LIN {X 0,Y 382.745,Z 469.054,A -85,B 0,C 180,E1 -14676.834,E2 -14676.834} C_VEL
LIN {X 0,Y 379.922,Z 466.3,A -85,B 0,C 180,E1 -14678.454,E2 -14678.454} C_VEL
LIN {X 0,Y 378.17,Z 464.212,A -85,B 0,C 180,E1 -14679.366,E2 -14679.366} C_VEL
LIN {X 0,Y 375.017,Z 462.339,A -85,B 0,C 180,E1 -14680.642,E2 -14680.642} C_VEL
LIN {X 0,Y 371.721,Z 459.429,A -85,B 0,C 180,E1 -14681.895,E2 -14681.895} C_VEL
LIN {X 0,Y 368.971,Z 456.558,A -85,B 0,C 180,E1 -14682.858,E2 -14682.858} C_VEL
LIN {X 0,Y 365.379,Z 453.694,A -85,B 0,C 180,E1 -14683.945,E2 -14683.945} C_VEL
LIN {X 0,Y 361.344,Z 449.449,A -85,B 0,C 180,E1 -14685.108,E2 -14685.108} C_VEL
LIN {X 0,Y 357.38,Z 445.807,A -85,B 0,C 180,E1 -14686.135,E2 -14686.135} C_VEL
LIN {X 0,Y 354.585,Z 442.813,A -85,B 0,C 180,E1 -14686.804,E2 -14686.804} C_VEL
LIN {X 0,Y 351.005,Z 439.151,A -85,B 0,C 180,E1 -14687.633,E2 -14687.633} C_VEL
LIN {X 0,Y 348.399,Z 436.221,A -85,B 0,C 180,E1 -14688.218,E2 -14688.218} C_VEL
LIN {X 0,Y 345.155,Z 432.375,A -85,B 0,C 180,E1 -14688.921,E2 -14688.921} C_VEL
LIN {X 0,Y 341.006,Z 427.451,A -85,B 0,C 180,E1 -14689.766,E2 -14689.766} C_VEL
LIN {X 0,Y 339.453,Z 425.497,A -85,B 0,C 180,E1 -14690.077,E2 -14690.077} C_VEL
LIN {X 0,Y 337.07,Z 422.222,A -85,B 0,C 180,E1 -14690.545,E2 -14690.545} C_VEL
LIN {X 0,Y 336.014,Z 420.806,A -85,B 0,C 180,E1 -14690.746,E2 -14690.746} C_VEL
LIN {X 0,Y 334.263,Z 418.461,A -85,B 0,C 180,E1 -14691.08,E2 -14691.08} C_VEL
LIN {X 0,Y 333.682,Z 416.42,A -85,B 0,C 180,E1 -14691.257,E2 -14691.257} C_VEL
LIN {X 0,Y 333.715,Z 416.415,A -85,B 0,C 180,E1 -14695.101,E2 -14695.101} C_VEL
LIN {X 0,Y 333.717,Z 416.414,A -85,B 0,C 180,E1 -14697.811,E2 -14697.811} C_VEL
LIN {X 0,Y 333.693,Z 416.42,A -85,B 0,C 180,E1 -14700.362,E2 -14700.362} C_VEL
LIN {X 0,Y 333.681,Z 416.42,A -85,B 0,C 180,E1 -14704.774,E2 -14704.774} C_VEL
LIN {X 0,Y 333.678,Z 416.42,A -85,B 0,C 180,E1 -14708.805,E2 -14708.805} C_VEL
LIN {X 0,Y 333.686,Z 416.421,A -85,B 0,C 180,E1 -14712.511,E2 -14712.511} C_VEL
LIN {X 0,Y 333.63,Z 416.426,A -85,B 0,C 180,E1 -14715.962,E2 -14715.962} C_VEL
LIN {X 0,Y 333.643,Z 416.422,A -85,B 0,C 180,E1 -14719.316,E2 -14719.316} C_VEL
LIN {X 0,Y 333.663,Z 416.419,A -85,B 0,C 180,E1 -14723.168,E2 -14723.168} C_VEL
LIN {X 0,Y 333.638,Z 416.423,A -85,B 0,C 180,E1 -14726.793,E2 -14726.793} C_VEL
LIN {X 0,Y 333.7,Z 416.417,A -85,B 0,C 180,E1 -14729.71,E2 -14729.71} C_VEL
LIN {X 0,Y 333.74,Z 416.412,A -85,B 0,C 180,E1 -14732.402,E2 -14732.402} C_VEL
LIN {X 0,Y 333.723,Z 416.411,A -85,B 0,C 180,E1 -14735.091,E2 -14735.091} C_VEL
LIN {X 0,Y 333.678,Z 416.417,A -85,B 0,C 180,E1 -14739.02,E2 -14739.02} C_VEL
LIN {X 0,Y 333.701,Z 416.414,A -85,B 0,C 180,E1 -14739.93,E2 -14739.93} C_VEL
LIN {X 0,Y 333.092,Z 416.492,A -85,B 0,C 180,E1 -14740.937,E2 -14740.937} C_VEL
LIN {X 0,Y 330.267,Z 416.843,A -85,B 0,C 180,E1 -14742.576,E2 -14742.576} C_VEL
LIN {X 0,Y 327.851,Z 417.148,A -85,B 0,C 180,E1 -14743.904,E2 -14743.904} C_VEL
LIN {X 0,Y 326.828,Z 417.27,A -85,B 0,C 180,E1 -14744.932,E2 -14744.932} C_VEL
LIN {X 0,Y 326.754,Z 417.28,A -85,B 0,C 180,E1 -14745.28,E2 -14745.28} C_VEL
LIN {X 0,Y 326.766,Z 417.278,A -85,B 0,C 180,E1 -14748.84,E2 -14748.84} C_VEL
LIN {X 0,Y 326.976,Z 417.253,A -85,B 0,C 180,E1 -14752.591,E2 -14752.591} C_VEL
LIN {X 0,Y 326.775,Z 417.277,A -85,B 0,C 180,E1 -14755.066,E2 -14755.066} C_VEL
LIN {X 0,Y 327.045,Z 417.244,A -85,B 0,C 180,E1 -14757.537,E2 -14757.537} C_VEL
LIN {X 0,Y 327.196,Z 417.226,A -85,B 0,C 180,E1 -14760.001,E2 -14760.001} C_VEL
LIN {X 0,Y 327.045,Z 417.244,A -85,B 0,C 180,E1 -14762.464,E2 -14762.464} C_VEL
LIN {X 0,Y 326.994,Z 417.251,A -85,B 0,C 180,E1 -14766.17,E2 -14766.17} C_VEL
LIN {X 0,Y 326.913,Z 417.261,A -85,B 0,C 180,E1 -14768.656,E2 -14768.656} C_VEL
LIN {X 0,Y 326.732,Z 417.283,A -85,B 0,C 180,E1 -14772.422,E2 -14772.422} C_VEL
LIN {X 0,Y 326.753,Z 417.282,A -85,B 0,C 180,E1 -14774.958,E2 -14774.958} C_VEL
LIN {X 0,Y 326.731,Z 417.285,A -85,B 0,C 180,E1 -14778.839,E2 -14778.839} C_VEL
LIN {X 0,Y 326.62,Z 417.299,A -85,B 0,C 180,E1 -14782.788,E2 -14782.788} C_VEL
LIN {X 0,Y 326.689,Z 417.291,A -85,B 0,C 180,E1 -14785.484,E2 -14785.484} C_VEL
LIN {X 0,Y 326.647,Z 417.297,A -85,B 0,C 180,E1 -14789.661,E2 -14789.661} C_VEL
LIN {X 0,Y 326.607,Z 417.301,A -85,B 0,C 180,E1 -14794.02,E2 -14794.02} C_VEL
LIN {X 0,Y 326.687,Z 417.697,A -85,B 0,C 180,E1 -14795.511,E2 -14795.511} C_VEL
LIN {X 0,Y 327.062,Z 420.418,A -85,B 0,C 180,E1 -14799.324,E2 -14799.324} C_VEL
LIN {X 0,Y 327.357,Z 422.259,A -85,B 0,C 180,E1 -14801.724,E2 -14801.724} C_VEL
LIN {X 0,Y 327.716,Z 424.981,A -85,B 0,C 180,E1 -14805.049,E2 -14805.049} C_VEL
LIN {X 0,Y 327.837,Z 427.974,A -85,B 0,C 180,E1 -14808.352,E2 -14808.352} C_VEL
LIN {X 0,Y 327.499,Z 431.094,A -85,B 0,C 180,E1 -14811.514,E2 -14811.514} C_VEL
LIN {X 0,Y 327.027,Z 434.493,A -85,B 0,C 180,E1 -14814.751,E2 -14814.751} C_VEL
LIN {X 0,Y 326.606,Z 437.456,A -85,B 0,C 180,E1 -14817.456,E2 -14817.456} C_VEL
LIN {X 0,Y 326.204,Z 440.67,A -85,B 0,C 180,E1 -14820.295,E2 -14820.295} C_VEL
LIN {X 0,Y 325.882,Z 443.915,A -85,B 0,C 180,E1 -14823.071,E2 -14823.071} C_VEL
LIN {X 0,Y 325.607,Z 447.183,A -85,B 0,C 180,E1 -14825.789,E2 -14825.789} C_VEL
LIN {X 0,Y 325.418,Z 449.412,A -85,B 0,C 180,E1 -14827.655,E2 -14827.655} C_VEL
LIN {X 0,Y 327.712,Z 459.083,A -85,B 0,C 180,E1 -14828.196,E2 -14828.196} C_VEL
LIN {X 0,Y 329.534,Z 468.228,A -85,B 0,C 180,E1 -14828.81,E2 -14828.81} C_VEL
LIN {X 0,Y 331.05,Z 477.851,A -85,B 0,C 180,E1 -14829.573,E2 -14829.573} C_VEL
LIN {X 0,Y 332.004,Z 486.455,A -85,B 0,C 180,E1 -14830.364,E2 -14830.364} C_VEL
LIN {X 0,Y 332.422,Z 491.382,A -85,B 0,C 180,E1 -14830.871,E2 -14830.871} C_VEL
LIN {X 0,Y 330.921,Z 503.575,A -85,B 0,C 180,E1 -14832.224,E2 -14832.224} C_VEL
LIN {X 0,Y 329.776,Z 512.454,A -85,B 0,C 180,E1 -14833.467,E2 -14833.467} C_VEL
LIN {X 0,Y 328.719,Z 520.466,A -85,B 0,C 180,E1 -14834.817,E2 -14834.817} C_VEL
LIN {X 0,Y 327.875,Z 526.671,A -85,B 0,C 180,E1 -14836.046,E2 -14836.046} C_VEL
LIN {X 0,Y 326.889,Z 533.209,A -85,B 0,C 180,E1 -14837.585,E2 -14837.585} C_VEL
LIN {X 0,Y 326.349,Z 537.716,A -85,B 0,C 180,E1 -14838.824,E2 -14838.824} C_VEL
LIN {X 0,Y 325.644,Z 543.21,A -85,B 0,C 180,E1 -14840.685,E2 -14840.685} C_VEL
LIN {X 0,Y 325.21,Z 547.538,A -85,B 0,C 180,E1 -14842.55,E2 -14842.55} C_VEL
LIN {X 0,Y 324.998,Z 550.39,A -85,B 0,C 180,E1 -14844.125,E2 -14844.125} C_VEL
LIN {X 0,Y 324.911,Z 553.099,A -85,B 0,C 180,E1 -14846.279,E2 -14846.279} C_VEL
LIN {X 0,Y 324.837,Z 554.158,A -85,B 0,C 180,E1 -14847.52,E2 -14847.52} C_VEL
LIN {X 0,Y 324.815,Z 554.747,A -85,B 0,C 180,E1 -14848.76,E2 -14848.76} C_VEL
LIN {X 0,Y 324.815,Z 554.747,A -85,B 0,C 180,E1 -14851.24,E2 -14851.24} C_VEL
LIN {X 0,Y 324.837,Z 554.158,A -85,B 0,C 180,E1 -14852.48,E2 -14852.48} C_VEL
LIN {X 0,Y 324.93,Z 551.71,A -85,B 0,C 180,E1 -14854.963,E2 -14854.963} C_VEL
LIN {X 0,Y 325.121,Z 548.758,A -85,B 0,C 180,E1 -14856.828,E2 -14856.828} C_VEL
LIN {X 0,Y 325.474,Z 544.766,A -85,B 0,C 180,E1 -14858.693,E2 -14858.693} C_VEL
LIN {X 0,Y 326.08,Z 539.634,A -85,B 0,C 180,E1 -14860.556,E2 -14860.556} C_VEL
LIN {X 0,Y 326.735,Z 534.368,A -85,B 0,C 180,E1 -14862.106,E2 -14862.106} C_VEL
LIN {X 0,Y 327.648,Z 528.05,A -85,B 0,C 180,E1 -14863.647,E2 -14863.647} C_VEL
LIN {X 0,Y 328.457,Z 522.096,A -85,B 0,C 180,E1 -14864.878,E2 -14864.878} C_VEL
LIN {X 0,Y 329.441,Z 515.168,A -85,B 0,C 180,E1 -14866.1,E2 -14866.1} C_VEL
LIN {X 0,Y 330.455,Z 506.983,A -85,B 0,C 180,E1 -14867.322,E2 -14867.322} C_VEL
LIN {X 0,Y 331.552,Z 498.472,A -85,B 0,C 180,E1 -14868.379,E2 -14868.379} C_VEL
LIN {X 0,Y 332.416,Z 491.388,A -85,B 0,C 180,E1 -14869.129,E2 -14869.129} C_VEL
LIN {X 0,Y 331.654,Z 482.381,A -85,B 0,C 180,E1 -14870.027,E2 -14870.027} C_VEL
LIN {X 0,Y 330.019,Z 471.038,A -85,B 0,C 180,E1 -14870.981,E2 -14870.981} C_VEL
LIN {X 0,Y 328.019,Z 460.532,A -85,B 0,C 180,E1 -14871.714,E2 -14871.714} C_VEL
LIN {X 0,Y 325.445,Z 449.866,A -85,B 0,C 180,E1 -14872.326,E2 -14872.326} C_VEL
LIN {X 0,Y 325.417,Z 449.413,A -85,B 0,C 180,E1 -14872.344,E2 -14872.344} C_VEL
LIN {X 0,Y 325.738,Z 445.556,A -85,B 0,C 180,E1 -14875.563,E2 -14875.563} C_VEL
LIN {X 0,Y 326.06,Z 442.285,A -85,B 0,C 180,E1 -14878.306,E2 -14878.306} C_VEL
LIN {X 0,Y 326.604,Z 437.433,A -85,B 0,C 180,E1 -14882.544,E2 -14882.544} C_VEL
LIN {X 0,Y 327.052,Z 434.248,A -85,B 0,C 180,E1 -14885.464,E2 -14885.464} C_VEL
LIN {X 0,Y 327.496,Z 431.094,A -85,B 0,C 180,E1 -14888.486,E2 -14888.486} C_VEL
LIN {X 0,Y 327.828,Z 427.973,A -85,B 0,C 180,E1 -14891.649,E2 -14891.649} C_VEL
LIN {X 0,Y 327.834,Z 426.427,A -85,B 0,C 180,E1 -14893.314,E2 -14893.314} C_VEL
LIN {X 0,Y 327.49,Z 423.385,A -85,B 0,C 180,E1 -14896.855,E2 -14896.855} C_VEL
LIN {X 0,Y 327.142,Z 421.004,A -85,B 0,C 180,E1 -14899.872,E2 -14899.872} C_VEL
LIN {X 0,Y 326.816,Z 418.723,A -85,B 0,C 180,E1 -14902.977,E2 -14902.977} C_VEL
LIN {X 0,Y 326.67,Z 417.471,A -85,B 0,C 180,E1 -14904.837,E2 -14904.837} C_VEL
LIN {X 0,Y 326.613,Z 417.301,A -85,B 0,C 180,E1 -14907.455,E2 -14907.455} C_VEL
LIN {X 0,Y 326.659,Z 417.295,A -85,B 0,C 180,E1 -14910.34,E2 -14910.34} C_VEL
LIN {X 0,Y 326.687,Z 417.293,A -85,B 0,C 180,E1 -14914.515,E2 -14914.515} C_VEL
LIN {X 0,Y 326.644,Z 417.299,A -85,B 0,C 180,E1 -14918.544,E2 -14918.544} C_VEL
LIN {X 0,Y 326.741,Z 417.284,A -85,B 0,C 180,E1 -14921.177,E2 -14921.177} C_VEL
LIN {X 0,Y 326.759,Z 417.28,A -85,B 0,C 180,E1 -14925.432,E2 -14925.432} C_VEL
LIN {X 0,Y 326.765,Z 417.282,A -85,B 0,C 180,E1 -14928.838,E2 -14928.838} C_VEL
LIN {X 0,Y 326.972,Z 417.258,A -85,B 0,C 180,E1 -14932.59,E2 -14932.59} C_VEL
LIN {X 0,Y 326.774,Z 417.279,A -85,B 0,C 180,E1 -14935.064,E2 -14935.064} C_VEL
LIN {X 0,Y 327.043,Z 417.244,A -85,B 0,C 180,E1 -14937.536,E2 -14937.536} C_VEL
LIN {X 0,Y 327.193,Z 417.226,A -85,B 0,C 180,E1 -14939.999,E2 -14939.999} C_VEL
LIN {X 0,Y 327.042,Z 417.244,A -85,B 0,C 180,E1 -14942.463,E2 -14942.463} C_VEL
LIN {X 0,Y 326.965,Z 417.254,A -85,B 0,C 180,E1 -14946.663,E2 -14946.663} C_VEL
LIN {X 0,Y 326.807,Z 417.275,A -85,B 0,C 180,E1 -14949.906,E2 -14949.906} C_VEL
LIN {X 0,Y 326.753,Z 417.282,A -85,B 0,C 180,E1 -14953.685,E2 -14953.685} C_VEL
LIN {X 0,Y 326.693,Z 417.289,A -85,B 0,C 180,E1 -14957.527,E2 -14957.527} C_VEL
LIN {X 0,Y 326.658,Z 417.296,A -85,B 0,C 180,E1 -14960.134,E2 -14960.134} C_VEL
LIN {X 0,Y 326.645,Z 417.297,A -85,B 0,C 180,E1 -14964.129,E2 -14964.129} C_VEL
LIN {X 0,Y 326.679,Z 417.29,A -85,B 0,C 180,E1 -14966.857,E2 -14966.857} C_VEL
LIN {X 0,Y 326.635,Z 417.295,A -85,B 0,C 180,E1 -14970.612,E2 -14970.612} C_VEL
LIN {X 0,Y 326.602,Z 417.303,A -85,B 0,C 180,E1 -14974.019,E2 -14974.019} C_VEL
LIN {X 0,Y 326.624,Z 417.297,A -85,B 0,C 180,E1 -14977.239,E2 -14977.239} C_VEL
LIN {X 0,Y 326.629,Z 417.297,A -85,B 0,C 180,E1 -14980.202,E2 -14980.202} C_VEL
LIN {X 0,Y 326.651,Z 417.296,A -85,B 0,C 180,E1 -14983.51,E2 -14983.51} C_VEL
LIN {X 0,Y 326.645,Z 417.295,A -85,B 0,C 180,E1 -14987.014,E2 -14987.014} C_VEL
LIN {X 0,Y 326.639,Z 417.295,A -85,B 0,C 180,E1 -14990.766,E2 -14990.766} C_VEL
LIN {X 0,Y 326.607,Z 417.299,A -85,B 0,C 180,E1 -14994.481,E2 -14994.481} C_VEL
LIN {X 0,Y 326.602,Z 417.305,A -85,B 0,C 180,E1 -14997.456,E2 -14997.456} C_VEL
LIN {X 0,Y 326.655,Z 417.293,A -85,B 0,C 180,E1 -15000.341,E2 -15000.341} C_VEL
LIN {X 0,Y 326.685,Z 417.29,A -85,B 0,C 180,E1 -15004.517,E2 -15004.517} C_VEL
LIN {X 0,Y 326.696,Z 417.417,A -85,B 0,C 180,E1 -15007.846,E2 -15007.846} C_VEL
LIN {X 0,Y 327.662,Z 420.137,A -85,B 0,C 180,E1 -15008.038,E2 -15008.038} C_VEL
LIN {X 0,Y 329.517,Z 422.658,A -85,B 0,C 180,E1 -15008.363,E2 -15008.363} C_VEL
LIN {X 0,Y 331.952,Z 426.11,A -85,B 0,C 180,E1 -15008.797,E2 -15008.797} C_VEL
LIN {X 0,Y 335.942,Z 431.227,A -85,B 0,C 180,E1 -15009.532,E2 -15009.532} C_VEL
LIN {X 0,Y 340.414,Z 436.618,A -85,B 0,C 180,E1 -15010.402,E2 -15010.402} C_VEL
LIN {X 0,Y 345.474,Z 442.37,A -85,B 0,C 180,E1 -15011.446,E2 -15011.446} C_VEL
LIN {X 0,Y 350.954,Z 448.276,A -85,B 0,C 180,E1 -15012.679,E2 -15012.679} C_VEL
LIN {X 0,Y 353.634,Z 450.976,A -85,B 0,C 180,E1 -15013.317,E2 -15013.317} C_VEL
LIN {X 0,Y 357.452,Z 454.808,A -85,B 0,C 180,E1 -15014.291,E2 -15014.291} C_VEL
LIN {X 0,Y 360.438,Z 457.628,A -85,B 0,C 180,E1 -15015.1,E2 -15015.1} C_VEL
LIN {X 0,Y 364.634,Z 461.722,A -85,B 0,C 180,E1 -15016.35,E2 -15016.35} C_VEL
LIN {X 0,Y 367.583,Z 464.131,A -85,B 0,C 180,E1 -15017.297,E2 -15017.297} C_VEL
LIN {X 0,Y 370.753,Z 467.398,A -85,B 0,C 180,E1 -15018.471,E2 -15018.471} C_VEL
LIN {X 0,Y 372.501,Z 468.815,A -85,B 0,C 180,E1 -15019.125,E2 -15019.125} C_VEL
LIN {X 0,Y 375.48,Z 470.669,A -85,B 0,C 180,E1 -15020.302,E2 -15020.302} C_VEL
LIN {X 0,Y 377.708,Z 473.025,A -85,B 0,C 180,E1 -15021.44,E2 -15021.44} C_VEL
LIN {X 0,Y 379.625,Z 475.01,A -85,B 0,C 180,E1 -15022.554,E2 -15022.554} C_VEL
LIN {X 0,Y 381.687,Z 476.586,A -85,B 0,C 180,E1 -15023.874,E2 -15023.874} C_VEL
LIN {X 0,Y 382.853,Z 477.331,A -85,B 0,C 180,E1 -15024.734,E2 -15024.734} C_VEL
LIN {X 0,Y 384.103,Z 477.928,A -85,B 0,C 180,E1 -15025.803,E2 -15025.803} C_VEL
LIN {X 0,Y 385.142,Z 478.17,A -85,B 0,C 180,E1 -15026.862,E2 -15026.862} C_VEL
LIN {X 0,Y 385.884,Z 478.349,A -85,B 0,C 180,E1 -15027.913,E2 -15027.913} C_VEL
LIN {X 0,Y 386.362,Z 478.4,A -85,B 0,C 180,E1 -15028.958,E2 -15028.958} C_VEL
LIN {X 0,Y 386.509,Z 478.455,A -85,B 0,C 180,E1 -15030,E2 -15030} C_VEL
LIN {X 0,Y 386.362,Z 478.373,A -85,B 0,C 180,E1 -15031.042,E2 -15031.042} C_VEL
LIN {X 0,Y 385.884,Z 478.332,A -85,B 0,C 180,E1 -15032.088,E2 -15032.088} C_VEL
LIN {X 0,Y 385.152,Z 478.141,A -85,B 0,C 180,E1 -15033.138,E2 -15033.138} C_VEL
LIN {X 0,Y 384.128,Z 477.899,A -85,B 0,C 180,E1 -15034.197,E2 -15034.197} C_VEL
LIN {X 0,Y 382.819,Z 477.344,A -85,B 0,C 180,E1 -15035.267,E2 -15035.267} C_VEL
LIN {X 0,Y 381.348,Z 476.385,A -85,B 0,C 180,E1 -15036.349,E2 -15036.349} C_VEL
LIN {X 0,Y 378.516,Z 473.912,A -85,B 0,C 180,E1 -15038.091,E2 -15038.091} C_VEL
LIN {X 0,Y 375.403,Z 470.647,A -85,B 0,C 180,E1 -15039.7,E2 -15039.7} C_VEL
LIN {X 0,Y 372.237,Z 468.61,A -85,B 0,C 180,E1 -15040.957,E2 -15040.957} C_VEL
LIN {X 0,Y 368.513,Z 465.192,A -85,B 0,C 180,E1 -15042.358,E2 -15042.358} C_VEL
LIN {X 0,Y 366.4,Z 463.033,A -85,B 0,C 180,E1 -15043.099,E2 -15043.099} C_VEL
LIN {X 0,Y 362.346,Z 459.667,A -85,B 0,C 180,E1 -15044.326,E2 -15044.326} C_VEL
LIN {X 0,Y 358.358,Z 455.575,A -85,B 0,C 180,E1 -15045.466,E2 -15045.466} C_VEL
LIN {X 0,Y 354.091,Z 451.552,A -85,B 0,C 180,E1 -15046.563,E2 -15046.563} C_VEL
LIN {X 0,Y 351.294,Z 448.583,A -85,B 0,C 180,E1 -15047.239,E2 -15047.239} C_VEL
LIN {X 0,Y 347.297,Z 444.338,A -85,B 0,C 180,E1 -15048.162,E2 -15048.162} C_VEL
LIN {X 0,Y 342.083,Z 438.594,A -85,B 0,C 180,E1 -15049.26,E2 -15049.26} C_VEL
LIN {X 0,Y 339.255,Z 435.384,A -85,B 0,C 180,E1 -15049.825,E2 -15049.825} C_VEL
LIN {X 0,Y 333.227,Z 427.768,A -85,B 0,C 180,E1 -15050.977,E2 -15050.977} C_VEL
LIN {X 0,Y 331.405,Z 425.511,A -85,B 0,C 180,E1 -15051.294,E2 -15051.294} C_VEL
LIN {X 0,Y 328.594,Z 421.346,A -85,B 0,C 180,E1 -15051.802,E2 -15051.802} C_VEL
LIN {X 0,Y 327.101,Z 418.951,A -85,B 0,C 180,E1 -15052.064,E2 -15052.064} C_VEL
LIN {X 0,Y 326.661,Z 417.295,A -85,B 0,C 180,E1 -15052.205,E2 -15052.205} C_VEL
LIN {X 0,Y 326.686,Z 417.29,A -85,B 0,C 180,E1 -15055.484,E2 -15055.484} C_VEL
LIN {X 0,Y 326.656,Z 417.293,A -85,B 0,C 180,E1 -15059.659,E2 -15059.659} C_VEL
LIN {X 0,Y 326.603,Z 417.301,A -85,B 0,C 180,E1 -15064.02,E2 -15064.02} C_VEL
LIN {X 0,Y 326.625,Z 417.297,A -85,B 0,C 180,E1 -15067.239,E2 -15067.239} C_VEL
LIN {X 0,Y 326.631,Z 417.3,A -85,B 0,C 180,E1 -15070.203,E2 -15070.203} C_VEL
LIN {X 0,Y 326.617,Z 417.297,A -85,B 0,C 180,E1 -15073.516,E2 -15073.516} C_VEL
LIN {X 0,Y 326.581,Z 417.302,A -85,B 0,C 180,E1 -15077.027,E2 -15077.027} C_VEL
LIN {X 0,Y 326.608,Z 417.299,A -85,B 0,C 180,E1 -15080.773,E2 -15080.773} C_VEL
LIN {X 0,Y 326.609,Z 417.301,A -85,B 0,C 180,E1 -15084.481,E2 -15084.481} C_VEL
LIN {X 0,Y 326.611,Z 417.299,A -85,B 0,C 180,E1 -15087.457,E2 -15087.457} C_VEL
LIN {X 0,Y 326.658,Z 417.295,A -85,B 0,C 180,E1 -15090.342,E2 -15090.342} C_VEL
LIN {X 0,Y 326.686,Z 417.288,A -85,B 0,C 180,E1 -15094.517,E2 -15094.517} C_VEL
LIN {X 0,Y 326.643,Z 417.294,A -85,B 0,C 180,E1 -15098.546,E2 -15098.546} C_VEL
LIN {X 0,Y 326.741,Z 417.282,A -85,B 0,C 180,E1 -15101.178,E2 -15101.178} C_VEL
LIN {X 0,Y 326.754,Z 417.28,A -85,B 0,C 180,E1 -15105.28,E2 -15105.28} C_VEL
LIN {X 0,Y 326.104,Z 417.365,A -85,B 0,C 180,E1 -15106.309,E2 -15106.309} C_VEL
LIN {X 0,Y 323.239,Z 417.722,A -85,B 0,C 180,E1 -15107.983,E2 -15107.983} C_VEL
LIN {X 0,Y 320.833,Z 418.019,A -85,B 0,C 180,E1 -15109.34,E2 -15109.34} C_VEL
LIN {X 0,Y 319.848,Z 418.14,A -85,B 0,C 180,E1 -15110.391,E2 -15110.391} C_VEL
LIN {X 0,Y 319.795,Z 418.146,A -85,B 0,C 180,E1 -15110.747,E2 -15110.747} C_VEL
LIN {X 0,Y 319.949,Z 418.133,A -85,B 0,C 180,E1 -15113.695,E2 -15113.695} C_VEL
LIN {X 0,Y 319.989,Z 418.121,A -85,B 0,C 180,E1 -15117.483,E2 -15117.483} C_VEL
LIN {X 0,Y 320.147,Z 418.103,A -85,B 0,C 180,E1 -15120.001,E2 -15120.001} C_VEL
LIN {X 0,Y 319.989,Z 418.123,A -85,B 0,C 180,E1 -15122.518,E2 -15122.518} C_VEL
LIN {X 0,Y 319.95,Z 418.128,A -85,B 0,C 180,E1 -15126.306,E2 -15126.306} C_VEL
LIN {X 0,Y 319.841,Z 418.142,A -85,B 0,C 180,E1 -15128.849,E2 -15128.849} C_VEL
LIN {X 0,Y 319.68,Z 418.162,A -85,B 0,C 180,E1 -15132.701,E2 -15132.701} C_VEL
LIN {X 0,Y 319.698,Z 418.164,A -85,B 0,C 180,E1 -15135.296,E2 -15135.296} C_VEL
LIN {X 0,Y 319.674,Z 418.168,A -85,B 0,C 180,E1 -15139.256,E2 -15139.256} C_VEL
LIN {X 0,Y 319.569,Z 418.181,A -85,B 0,C 180,E1 -15143.32,E2 -15143.32} C_VEL
LIN {X 0,Y 319.618,Z 418.169,A -85,B 0,C 180,E1 -15146.09,E2 -15146.09} C_VEL
LIN {X 0,Y 319.58,Z 418.179,A -85,B 0,C 180,E1 -15148.935,E2 -15148.935} C_VEL
LIN {X 0,Y 319.53,Z 418.184,A -85,B 0,C 180,E1 -15151.863,E2 -15151.863} C_VEL
LIN {X 0,Y 319.629,Z 418.434,A -85,B 0,C 180,E1 -15154.869,E2 -15154.869} C_VEL
LIN {X 0,Y 319.931,Z 420.541,A -85,B 0,C 180,E1 -15157.959,E2 -15157.959} C_VEL
LIN {X 0,Y 320.347,Z 423.316,A -85,B 0,C 180,E1 -15161.763,E2 -15161.763} C_VEL
LIN {X 0,Y 320.69,Z 426.349,A -85,B 0,C 180,E1 -15165.47,E2 -15165.47} C_VEL
LIN {X 0,Y 320.813,Z 428.725,A -85,B 0,C 180,E1 -15168.146,E2 -15168.146} C_VEL
LIN {X 0,Y 320.593,Z 430.992,A -85,B 0,C 180,E1 -15170.526,E2 -15170.526} C_VEL
LIN {X 0,Y 320.012,Z 434.863,A -85,B 0,C 180,E1 -15174.35,E2 -15174.35} C_VEL
LIN {X 0,Y 319.679,Z 437.315,A -85,B 0,C 180,E1 -15176.66,E2 -15176.66} C_VEL
LIN {X 0,Y 319.254,Z 440.531,A -85,B 0,C 180,E1 -15179.581,E2 -15179.581} C_VEL
LIN {X 0,Y 318.898,Z 443.74,A -85,B 0,C 180,E1 -15182.432,E2 -15182.432} C_VEL
LIN {X 0,Y 318.576,Z 446.987,A -85,B 0,C 180,E1 -15185.219,E2 -15185.219} C_VEL
LIN {X 0,Y 318.398,Z 449.196,A -85,B 0,C 180,E1 -15187.115,E2 -15187.115} C_VEL
LIN {X 0,Y 321.885,Z 464.143,A -85,B 0,C 180,E1 -15188.037,E2 -15188.037} C_VEL
LIN {X 0,Y 323.959,Z 476.646,A -85,B 0,C 180,E1 -15189.025,E2 -15189.025} C_VEL
LIN {X 0,Y 325.107,Z 486.237,A -85,B 0,C 180,E1 -15189.929,E2 -15189.929} C_VEL
LIN {X 0,Y 325.549,Z 492.782,A -85,B 0,C 180,E1 -15190.615,E2 -15190.615} C_VEL
LIN {X 0,Y 324.16,Z 503.364,A -85,B 0,C 180,E1 -15191.841,E2 -15191.841} C_VEL
LIN {X 0,Y 323.051,Z 511.495,A -85,B 0,C 180,E1 -15192.986,E2 -15192.986} C_VEL
LIN {X 0,Y 321.848,Z 520.28,A -85,B 0,C 180,E1 -15194.49,E2 -15194.49} C_VEL
LIN {X 0,Y 320.978,Z 526.46,A -85,B 0,C 180,E1 -15195.74,E2 -15195.74} C_VEL
LIN {X 0,Y 319.931,Z 532.997,A -85,B 0,C 180,E1 -15197.31,E2 -15197.31} C_VEL
LIN {X 0,Y 319.332,Z 537.503,A -85,B 0,C 180,E1 -15198.575,E2 -15198.575} C_VEL
LIN {X 0,Y 318.624,Z 542.998,A -85,B 0,C 180,E1 -15200.478,E2 -15200.478} C_VEL
LIN {X 0,Y 318.145,Z 547.326,A -85,B 0,C 180,E1 -15202.383,E2 -15202.383} C_VEL
LIN {X 0,Y 317.889,Z 550.475,A -85,B 0,C 180,E1 -15204.203,E2 -15204.203} C_VEL
LIN {X 0,Y 317.82,Z 552.888,A -85,B 0,C 180,E1 -15206.196,E2 -15206.196} C_VEL
LIN {X 0,Y 317.76,Z 553.947,A -85,B 0,C 180,E1 -15207.464,E2 -15207.464} C_VEL
LIN {X 0,Y 317.728,Z 554.536,A -85,B 0,C 180,E1 -15208.732,E2 -15208.732} C_VEL
LIN {X 0,Y 317.728,Z 554.536,A -85,B 0,C 180,E1 -15211.267,E2 -15211.267} C_VEL
LIN {X 0,Y 317.76,Z 553.947,A -85,B 0,C 180,E1 -15212.535,E2 -15212.535} C_VEL
LIN {X 0,Y 317.846,Z 551.498,A -85,B 0,C 180,E1 -15215.074,E2 -15215.074} C_VEL
LIN {X 0,Y 318.064,Z 548.546,A -85,B 0,C 180,E1 -15216.98,E2 -15216.98} C_VEL
LIN {X 0,Y 318.425,Z 544.554,A -85,B 0,C 180,E1 -15218.887,E2 -15218.887} C_VEL
LIN {X 0,Y 319.065,Z 539.421,A -85,B 0,C 180,E1 -15220.791,E2 -15220.791} C_VEL
LIN {X 0,Y 319.772,Z 534.156,A -85,B 0,C 180,E1 -15222.373,E2 -15222.373} C_VEL
LIN {X 0,Y 320.739,Z 527.838,A -85,B 0,C 180,E1 -15223.947,E2 -15223.947} C_VEL
LIN {X 0,Y 321.572,Z 521.883,A -85,B 0,C 180,E1 -15225.204,E2 -15225.204} C_VEL
LIN {X 0,Y 322.651,Z 514.177,A -85,B 0,C 180,E1 -15226.58,E2 -15226.58} C_VEL
LIN {X 0,Y 323.653,Z 506.771,A -85,B 0,C 180,E1 -15227.698,E2 -15227.698} C_VEL
LIN {X 0,Y 324.792,Z 498.259,A -85,B 0,C 180,E1 -15228.776,E2 -15228.776} C_VEL
LIN {X 0,Y 325.587,Z 491.172,A -85,B 0,C 180,E1 -15229.546,E2 -15229.546} C_VEL
LIN {X 0,Y 324.515,Z 480.611,A -85,B 0,C 180,E1 -15230.613,E2 -15230.613} C_VEL
LIN {X 0,Y 323.108,Z 471.159,A -85,B 0,C 180,E1 -15231.429,E2 -15231.429} C_VEL
LIN {X 0,Y 321.092,Z 460.665,A -85,B 0,C 180,E1 -15232.19,E2 -15232.19} C_VEL
LIN {X 0,Y 318.429,Z 449.812,A -85,B 0,C 180,E1 -15232.84,E2 -15232.84} C_VEL
LIN {X 0,Y 318.38,Z 449.164,A -85,B 0,C 180,E1 -15232.914,E2 -15232.914} C_VEL
LIN {X 0,Y 318.721,Z 445.358,A -85,B 0,C 180,E1 -15236.168,E2 -15236.168} C_VEL
LIN {X 0,Y 319.036,Z 442.114,A -85,B 0,C 180,E1 -15238.988,E2 -15238.988} C_VEL
LIN {X 0,Y 319.407,Z 438.9,A -85,B 0,C 180,E1 -15241.875,E2 -15241.875} C_VEL
LIN {X 0,Y 320.008,Z 434.861,A -85,B 0,C 180,E1 -15245.649,E2 -15245.649} C_VEL
LIN {X 0,Y 320.592,Z 430.991,A -85,B 0,C 180,E1 -15249.474,E2 -15249.474} C_VEL
LIN {X 0,Y 320.804,Z 427.883,A -85,B 0,C 180,E1 -15252.775,E2 -15252.775} C_VEL
LIN {X 0,Y 320.513,Z 424.817,A -85,B 0,C 180,E1 -15256.351,E2 -15256.351} C_VEL
LIN {X 0,Y 320.29,Z 422.871,A -85,B 0,C 180,E1 -15258.83,E2 -15258.83} C_VEL
LIN {X 0,Y 319.862,Z 420.357,A -85,B 0,C 180,E1 -15262.277,E2 -15262.277} C_VEL
LIN {X 0,Y 319.637,Z 418.421,A -85,B 0,C 180,E1 -15265.132,E2 -15265.132} C_VEL
LIN {X 0,Y 319.536,Z 418.182,A -85,B 0,C 180,E1 -15268.138,E2 -15268.138} C_VEL
LIN {X 0,Y 319.614,Z 418.171,A -85,B 0,C 180,E1 -15271.587,E2 -15271.587} C_VEL
LIN {X 0,Y 319.601,Z 418.174,A -85,B 0,C 180,E1 -15275.303,E2 -15275.303} C_VEL
LIN {X 0,Y 319.594,Z 418.174,A -85,B 0,C 180,E1 -15278.047,E2 -15278.047} C_VEL
LIN {X 0,Y 319.685,Z 418.165,A -85,B 0,C 180,E1 -15280.961,E2 -15280.961} C_VEL
LIN {X 0,Y 319.726,Z 418.156,A -85,B 0,C 180,E1 -15285.275,E2 -15285.275} C_VEL
LIN {X 0,Y 319.753,Z 418.153,A -85,B 0,C 180,E1 -15289.872,E2 -15289.872} C_VEL
LIN {X 0,Y 319.929,Z 418.135,A -85,B 0,C 180,E1 -15292.425,E2 -15292.425} C_VEL
LIN {X 0,Y 319.743,Z 418.155,A -85,B 0,C 180,E1 -15294.955,E2 -15294.955} C_VEL
LIN {X 0,Y 319.987,Z 418.123,A -85,B 0,C 180,E1 -15297.482,E2 -15297.482} C_VEL
LIN {X 0,Y 320.144,Z 418.104,A -85,B 0,C 180,E1 -15299.999,E2 -15299.999} C_VEL
LIN {X 0,Y 319.986,Z 418.122,A -85,B 0,C 180,E1 -15302.517,E2 -15302.517} C_VEL
LIN {X 0,Y 319.925,Z 418.133,A -85,B 0,C 180,E1 -15306.654,E2 -15306.654} C_VEL
LIN {X 0,Y 319.751,Z 418.156,A -85,B 0,C 180,E1 -15310.127,E2 -15310.127} C_VEL
LIN {X 0,Y 319.725,Z 418.155,A -85,B 0,C 180,E1 -15314.724,E2 -15314.724} C_VEL
LIN {X 0,Y 319.683,Z 418.16,A -85,B 0,C 180,E1 -15319.037,E2 -15319.037} C_VEL
LIN {X 0,Y 319.564,Z 418.176,A -85,B 0,C 180,E1 -15323.319,E2 -15323.319} C_VEL
LIN {X 0,Y 319.628,Z 418.173,A -85,B 0,C 180,E1 -15326.088,E2 -15326.088} C_VEL
LIN {X 0,Y 319.583,Z 418.173,A -85,B 0,C 180,E1 -15328.933,E2 -15328.933} C_VEL
LIN {X 0,Y 319.532,Z 418.185,A -85,B 0,C 180,E1 -15331.861,E2 -15331.861} C_VEL
LIN {X 0,Y 319.574,Z 418.178,A -85,B 0,C 180,E1 -15335.543,E2 -15335.543} C_VEL
LIN {X 0,Y 319.594,Z 418.176,A -85,B 0,C 180,E1 -15338.004,E2 -15338.004} C_VEL
LIN {X 0,Y 319.595,Z 418.176,A -85,B 0,C 180,E1 -15341.612,E2 -15341.612} C_VEL
LIN {X 0,Y 319.639,Z 418.168,A -85,B 0,C 180,E1 -15345.285,E2 -15345.285} C_VEL
LIN {X 0,Y 319.577,Z 418.174,A -85,B 0,C 180,E1 -15348.721,E2 -15348.721} C_VEL
LIN {X 0,Y 319.592,Z 418.173,A -85,B 0,C 180,E1 -15352.339,E2 -15352.339} C_VEL
LIN {X 0,Y 319.554,Z 418.179,A -85,B 0,C 180,E1 -15355.124,E2 -15355.124} C_VEL
LIN {X 0,Y 319.564,Z 418.178,A -85,B 0,C 180,E1 -15359.058,E2 -15359.058} C_VEL
LIN {X 0,Y 319.603,Z 418.172,A -85,B 0,C 180,E1 -15362.498,E2 -15362.498} C_VEL
LIN {X 0,Y 319.6,Z 418.176,A -85,B 0,C 180,E1 -15365.304,E2 -15365.304} C_VEL
LIN {X 0,Y 319.568,Z 418.179,A -85,B 0,C 180,E1 -15367.015,E2 -15367.015} C_VEL
LIN {X 0,Y 320.7,Z 421.226,A -85,B 0,C 180,E1 -15367.231,E2 -15367.231} C_VEL
LIN {X 0,Y 322.464,Z 423.884,A -85,B 0,C 180,E1 -15367.502,E2 -15367.502} C_VEL
LIN {X 0,Y 327.551,Z 431.069,A -85,B 0,C 180,E1 -15368.33,E2 -15368.33} C_VEL
LIN {X 0,Y 332.156,Z 436.822,A -85,B 0,C 180,E1 -15369.15,E2 -15369.15} C_VEL
LIN {X 0,Y 336.809,Z 442.321,A -85,B 0,C 180,E1 -15370.04,E2 -15370.04} C_VEL
LIN {X 0,Y 341.976,Z 448.216,A -85,B 0,C 180,E1 -15371.106,E2 -15371.106} C_VEL
LIN {X 0,Y 347.397,Z 454.063,A -85,B 0,C 180,E1 -15372.335,E2 -15372.335} C_VEL
LIN {X 0,Y 350.406,Z 457.126,A -85,B 0,C 180,E1 -15373.057,E2 -15373.057} C_VEL
LIN {X 0,Y 354.457,Z 461.123,A -85,B 0,C 180,E1 -15374.098,E2 -15374.098} C_VEL
LIN {X 0,Y 356.924,Z 463.403,A -85,B 0,C 180,E1 -15374.757,E2 -15374.757} C_VEL
LIN {X 0,Y 361.794,Z 468.184,A -85,B 0,C 180,E1 -15376.23,E2 -15376.23} C_VEL
LIN {X 0,Y 364.939,Z 470.846,A -85,B 0,C 180,E1 -15377.234,E2 -15377.234} C_VEL
LIN {X 0,Y 367.796,Z 473.747,A -85,B 0,C 180,E1 -15378.304,E2 -15378.304} C_VEL
LIN {X 0,Y 371.446,Z 476.364,A -85,B 0,C 180,E1 -15379.693,E2 -15379.693} C_VEL
LIN {X 0,Y 373.743,Z 478.206,A -85,B 0,C 180,E1 -15380.711,E2 -15380.711} C_VEL
LIN {X 0,Y 376.856,Z 481.513,A -85,B 0,C 180,E1 -15382.499,E2 -15382.499} C_VEL
LIN {X 0,Y 378.598,Z 482.895,A -85,B 0,C 180,E1 -15383.606,E2 -15383.606} C_VEL
LIN {X 0,Y 380.812,Z 484.209,A -85,B 0,C 180,E1 -15385.255,E2 -15385.255} C_VEL
LIN {X 0,Y 382.489,Z 484.732,A -85,B 0,C 180,E1 -15386.84,E2 -15386.84} C_VEL
LIN {X 0,Y 383.25,Z 484.938,A -85,B 0,C 180,E1 -15387.898,E2 -15387.898} C_VEL
LIN {X 0,Y 383.748,Z 484.979,A -85,B 0,C 180,E1 -15388.951,E2 -15388.951} C_VEL
LIN {X 0,Y 383.889,Z 485.041,A -85,B 0,C 180,E1 -15390,E2 -15390} C_VEL
LIN {X 0,Y 383.738,Z 484.972,A -85,B 0,C 180,E1 -15391.05,E2 -15391.05} C_VEL
LIN {X 0,Y 383.246,Z 484.925,A -85,B 0,C 180,E1 -15392.102,E2 -15392.102} C_VEL
LIN {X 0,Y 382.496,Z 484.712,A -85,B 0,C 180,E1 -15393.16,E2 -15393.16} C_VEL
LIN {X 0,Y 380.815,Z 484.181,A -85,B 0,C 180,E1 -15394.75,E2 -15394.75} C_VEL
LIN {X 0,Y 378.587,Z 482.896,A -85,B 0,C 180,E1 -15396.395,E2 -15396.395} C_VEL
LIN {X 0,Y 376.106,Z 480.765,A -85,B 0,C 180,E1 -15397.964,E2 -15397.964} C_VEL
LIN {X 0,Y 372.704,Z 477.231,A -85,B 0,C 180,E1 -15399.771,E2 -15399.771} C_VEL
LIN {X 0,Y 369.74,Z 475.312,A -85,B 0,C 180,E1 -15400.958,E2 -15400.958} C_VEL
LIN {X 0,Y 366.53,Z 472.52,A -85,B 0,C 180,E1 -15402.176,E2 -15402.176} C_VEL
LIN {X 0,Y 361.787,Z 468.158,A -85,B 0,C 180,E1 -15403.766,E2 -15403.766} C_VEL
LIN {X 0,Y 358.463,Z 465.139,A -85,B 0,C 180,E1 -15404.766,E2 -15404.766} C_VEL
LIN {X 0,Y 355.444,Z 461.927,A -85,B 0,C 180,E1 -15405.646,E2 -15405.646} C_VEL
LIN {X 0,Y 350.779,Z 457.592,A -85,B 0,C 180,E1 -15406.845,E2 -15406.845} C_VEL
LIN {X 0,Y 348.046,Z 454.7,A -85,B 0,C 180,E1 -15407.515,E2 -15407.515} C_VEL
LIN {X 0,Y 343.645,Z 450.019,A -85,B 0,C 180,E1 -15408.527,E2 -15408.527} C_VEL
LIN {X 0,Y 338.288,Z 444.098,A -85,B 0,C 180,E1 -15409.656,E2 -15409.656} C_VEL
LIN {X 0,Y 333.052,Z 437.879,A -85,B 0,C 180,E1 -15410.684,E2 -15410.684} C_VEL
LIN {X 0,Y 328.939,Z 432.779,A -85,B 0,C 180,E1 -15411.432,E2 -15411.432} C_VEL
LIN {X 0,Y 325.207,Z 427.862,A -85,B 0,C 180,E1 -15412.063,E2 -15412.063} C_VEL
LIN {X 0,Y 322.039,Z 423.1,A -85,B 0,C 180,E1 -15412.571,E2 -15412.571} C_VEL
LIN {X 0,Y 319.97,Z 419.804,A -85,B 0,C 180,E1 -15412.881,E2 -15412.881} C_VEL
LIN {X 0,Y 319.578,Z 418.178,A -85,B 0,C 180,E1 -15413.004,E2 -15413.004} C_VEL
LIN {X 0,Y 319.631,Z 418.17,A -85,B 0,C 180,E1 -15416.088,E2 -15416.088} C_VEL
LIN {X 0,Y 319.586,Z 418.176,A -85,B 0,C 180,E1 -15418.934,E2 -15418.934} C_VEL
LIN {X 0,Y 319.528,Z 418.182,A -85,B 0,C 180,E1 -15421.862,E2 -15421.862} C_VEL
LIN {X 0,Y 319.576,Z 418.175,A -85,B 0,C 180,E1 -15425.543,E2 -15425.543} C_VEL
LIN {X 0,Y 319.596,Z 418.174,A -85,B 0,C 180,E1 -15428.005,E2 -15428.005} C_VEL
LIN {X 0,Y 319.593,Z 418.173,A -85,B 0,C 180,E1 -15431.612,E2 -15431.612} C_VEL
LIN {X 0,Y 319.538,Z 418.179,A -85,B 0,C 180,E1 -15435.267,E2 -15435.267} C_VEL
LIN {X 0,Y 319.524,Z 418.182,A -85,B 0,C 180,E1 -15438.712,E2 -15438.712} C_VEL
LIN {X 0,Y 319.574,Z 418.179,A -85,B 0,C 180,E1 -15442.344,E2 -15442.344} C_VEL
LIN {X 0,Y 319.556,Z 418.177,A -85,B 0,C 180,E1 -15445.124,E2 -15445.124} C_VEL
LIN {X 0,Y 319.571,Z 418.175,A -85,B 0,C 180,E1 -15449.057,E2 -15449.057} C_VEL
LIN {X 0,Y 319.605,Z 418.172,A -85,B 0,C 180,E1 -15452.499,E2 -15452.499} C_VEL
LIN {X 0,Y 319.601,Z 418.17,A -85,B 0,C 180,E1 -15455.305,E2 -15455.305} C_VEL
LIN {X 0,Y 319.593,Z 418.176,A -85,B 0,C 180,E1 -15458.048,E2 -15458.048} C_VEL
LIN {X 0,Y 319.686,Z 418.16,A -85,B 0,C 180,E1 -15460.963,E2 -15460.963} C_VEL
LIN {X 0,Y 319.728,Z 418.155,A -85,B 0,C 180,E1 -15465.277,E2 -15465.277} C_VEL
LIN {X 0,Y 319.754,Z 418.155,A -85,B 0,C 180,E1 -15469.873,E2 -15469.873} C_VEL
LIN {X 0,Y 319.795,Z 418.146,A -85,B 0,C 180,E1 -15470.747,E2 -15470.747} C_VEL
LIN {X 0,Y 319.519,Z 418.183,A -85,B 0,C 180,E1 -15471.45,E2 -15471.45} C_VEL
LIN {X 0,Y 318.158,Z 418.354,A -85,B 0,C 180,E1 -15472.487,E2 -15472.487} C_VEL
LIN {X 0,Y 313.746,Z 418.902,A -85,B 0,C 180,E1 -15474.893,E2 -15474.893} C_VEL
LIN {X 0,Y 312.757,Z 419.022,A -85,B 0,C 180,E1 -15475.969,E2 -15475.969} C_VEL
LIN {X 0,Y 312.719,Z 419.024,A -85,B 0,C 180,E1 -15476.333,E2 -15476.333} C_VEL
LIN {X 0,Y 312.988,Z 418.988,A -85,B 0,C 180,E1 -15478.714,E2 -15478.714} C_VEL
LIN {X 0,Y 312.988,Z 418.996,A -85,B 0,C 180,E1 -15481.287,E2 -15481.287} C_VEL
LIN {X 0,Y 312.716,Z 419.031,A -85,B 0,C 180,E1 -15485.158,E2 -15485.158} C_VEL
LIN {X 0,Y 312.872,Z 419.013,A -85,B 0,C 180,E1 -15487.746,E2 -15487.746} C_VEL
LIN {X 0,Y 312.667,Z 419.039,A -85,B 0,C 180,E1 -15491.672,E2 -15491.672} C_VEL
LIN {X 0,Y 312.699,Z 419.033,A -85,B 0,C 180,E1 -15494.888,E2 -15494.888} C_VEL
LIN {X 0,Y 312.629,Z 419.045,A -85,B 0,C 180,E1 -15499.237,E2 -15499.237} C_VEL
LIN {X 0,Y 312.545,Z 419.052,A -85,B 0,C 180,E1 -15502.79,E2 -15502.79} C_VEL
LIN {X 0,Y 312.596,Z 419.044,A -85,B 0,C 180,E1 -15505.934,E2 -15505.934} C_VEL
LIN {X 0,Y 312.538,Z 419.055,A -85,B 0,C 180,E1 -15509.651,E2 -15509.651} C_VEL
LIN {X 0,Y 312.529,Z 419.057,A -85,B 0,C 180,E1 -15513.692,E2 -15513.692} C_VEL
LIN {X 0,Y 312.703,Z 420.307,A -85,B 0,C 180,E1 -15515.993,E2 -15515.993} C_VEL
LIN {X 0,Y 312.986,Z 422.321,A -85,B 0,C 180,E1 -15518.957,E2 -15518.957} C_VEL
LIN {X 0,Y 313.385,Z 424.789,A -85,B 0,C 180,E1 -15522.283,E2 -15522.283} C_VEL
LIN {X 0,Y 313.69,Z 427.801,A -85,B 0,C 180,E1 -15526.01,E2 -15526.01} C_VEL
LIN {X 0,Y 313.762,Z 429.338,A -85,B 0,C 180,E1 -15527.781,E2 -15527.781} C_VEL
LIN {X 0,Y 313.438,Z 432.443,A -85,B 0,C 180,E1 -15531.111,E2 -15531.111} C_VEL
LIN {X 0,Y 312.985,Z 435.587,A -85,B 0,C 180,E1 -15534.28,E2 -15534.28} C_VEL
LIN {X 0,Y 312.48,Z 438.77,A -85,B 0,C 180,E1 -15537.331,E2 -15537.331} C_VEL
LIN {X 0,Y 311.903,Z 443.571,A -85,B 0,C 180,E1 -15541.759,E2 -15541.759} C_VEL
LIN {X 0,Y 311.566,Z 446.813,A -85,B 0,C 180,E1 -15544.622,E2 -15544.622} C_VEL
LIN {X 0,Y 311.347,Z 449.115,A -85,B 0,C 180,E1 -15546.595,E2 -15546.595} C_VEL
LIN {X 0,Y 313.76,Z 458.95,A -85,B 0,C 180,E1 -15547.189,E2 -15547.189} C_VEL
LIN {X 0,Y 315.688,Z 468.061,A -85,B 0,C 180,E1 -15547.851,E2 -15547.851} C_VEL
LIN {X 0,Y 317.241,Z 478.051,A -85,B 0,C 180,E1 -15548.696,E2 -15548.696} C_VEL
LIN {X 0,Y 318.33,Z 487.661,A -85,B 0,C 180,E1 -15549.652,E2 -15549.652} C_VEL
LIN {X 0,Y 318.779,Z 492.568,A -85,B 0,C 180,E1 -15550.186,E2 -15550.186} C_VEL
LIN {X 0,Y 317.408,Z 503.152,A -85,B 0,C 180,E1 -15551.441,E2 -15551.441} C_VEL
LIN {X 0,Y 316.309,Z 510.899,A -85,B 0,C 180,E1 -15552.545,E2 -15552.545} C_VEL
LIN {X 0,Y 315.211,Z 518.816,A -85,B 0,C 180,E1 -15553.899,E2 -15553.899} C_VEL
LIN {X 0,Y 314.072,Z 526.248,A -85,B 0,C 180,E1 -15555.419,E2 -15555.419} C_VEL
LIN {X 0,Y 312.989,Z 532.785,A -85,B 0,C 180,E1 -15557.024,E2 -15557.024} C_VEL
LIN {X 0,Y 312.328,Z 537.29,A -85,B 0,C 180,E1 -15558.316,E2 -15558.316} C_VEL
LIN {X 0,Y 311.586,Z 542.786,A -85,B 0,C 180,E1 -15560.26,E2 -15560.26} C_VEL
LIN {X 0,Y 311.071,Z 547.114,A -85,B 0,C 180,E1 -15562.209,E2 -15562.209} C_VEL
LIN {X 0,Y 310.899,Z 549.484,A -85,B 0,C 180,E1 -15563.51,E2 -15563.51} C_VEL
LIN {X 0,Y 310.764,Z 551.286,A -85,B 0,C 180,E1 -15564.81,E2 -15564.81} C_VEL
LIN {X 0,Y 310.684,Z 553.736,A -85,B 0,C 180,E1 -15567.407,E2 -15567.407} C_VEL
LIN {X 0,Y 310.643,Z 554.325,A -85,B 0,C 180,E1 -15568.703,E2 -15568.703} C_VEL
LIN {X 0,Y 310.643,Z 554.325,A -85,B 0,C 180,E1 -15571.296,E2 -15571.296} C_VEL
LIN {X 0,Y 310.684,Z 553.736,A -85,B 0,C 180,E1 -15572.593,E2 -15572.593} C_VEL
LIN {X 0,Y 310.766,Z 551.286,A -85,B 0,C 180,E1 -15575.19,E2 -15575.19} C_VEL
LIN {X 0,Y 311.001,Z 548.334,A -85,B 0,C 180,E1 -15577.139,E2 -15577.139} C_VEL
LIN {X 0,Y 311.396,Z 544.342,A -85,B 0,C 180,E1 -15579.09,E2 -15579.09} C_VEL
LIN {X 0,Y 312.061,Z 539.209,A -85,B 0,C 180,E1 -15581.036,E2 -15581.036} C_VEL
LIN {X 0,Y 312.79,Z 533.943,A -85,B 0,C 180,E1 -15582.654,E2 -15582.654} C_VEL
LIN {X 0,Y 313.826,Z 527.626,A -85,B 0,C 180,E1 -15584.261,E2 -15584.261} C_VEL
LIN {X 0,Y 314.707,Z 521.672,A -85,B 0,C 180,E1 -15585.544,E2 -15585.544} C_VEL
LIN {X 0,Y 315.715,Z 514.742,A -85,B 0,C 180,E1 -15586.821,E2 -15586.821} C_VEL
LIN {X 0,Y 316.891,Z 506.56,A -85,B 0,C 180,E1 -15588.088,E2 -15588.088} C_VEL
LIN {X 0,Y 318.053,Z 498.047,A -85,B 0,C 180,E1 -15589.189,E2 -15589.189} C_VEL
LIN {X 0,Y 318.761,Z 492.573,A -85,B 0,C 180,E1 -15589.814,E2 -15589.814} C_VEL
LIN {X 0,Y 317.74,Z 481.474,A -85,B 0,C 180,E1 -15590.983,E2 -15590.983} C_VEL
LIN {X 0,Y 316.156,Z 470.613,A -85,B 0,C 180,E1 -15591.946,E2 -15591.946} C_VEL
LIN {X 0,Y 314.066,Z 460.24,A -85,B 0,C 180,E1 -15592.724,E2 -15592.724} C_VEL
LIN {X 0,Y 311.393,Z 449.712,A -85,B 0,C 180,E1 -15593.382,E2 -15593.382} C_VEL
LIN {X 0,Y 311.33,Z 449.004,A -85,B 0,C 180,E1 -15593.431,E2 -15593.431} C_VEL
LIN {X 0,Y 311.708,Z 445.159,A -85,B 0,C 180,E1 -15596.803,E2 -15596.803} C_VEL
LIN {X 0,Y 312.048,Z 441.943,A -85,B 0,C 180,E1 -15599.701,E2 -15599.701} C_VEL
LIN {X 0,Y 312.63,Z 437.653,A -85,B 0,C 180,E1 -15603.718,E2 -15603.718} C_VEL
LIN {X 0,Y 313.183,Z 434.007,A -85,B 0,C 180,E1 -15607.292,E2 -15607.292} C_VEL
LIN {X 0,Y 313.65,Z 430.884,A -85,B 0,C 180,E1 -15610.526,E2 -15610.526} C_VEL
LIN {X 0,Y 313.757,Z 429.229,A -85,B 0,C 180,E1 -15612.337,E2 -15612.337} C_VEL
LIN {X 0,Y 313.532,Z 426.249,A -85,B 0,C 180,E1 -15615.831,E2 -15615.831} C_VEL
LIN {X 0,Y 313.168,Z 423.492,A -85,B 0,C 180,E1 -15619.397,E2 -15619.397} C_VEL
LIN {X 0,Y 312.802,Z 421.23,A -85,B 0,C 180,E1 -15622.653,E2 -15622.653} C_VEL
LIN {X 0,Y 312.543,Z 419.16,A -85,B 0,C 180,E1 -15625.794,E2 -15625.794} C_VEL
LIN {X 0,Y 312.526,Z 419.058,A -85,B 0,C 180,E1 -15628.853,E2 -15628.853} C_VEL
LIN {X 0,Y 312.572,Z 419.048,A -85,B 0,C 180,E1 -15631.824,E2 -15631.824} C_VEL
LIN {X 0,Y 312.582,Z 419.052,A -85,B 0,C 180,E1 -15634.71,E2 -15634.71} C_VEL
LIN {X 0,Y 312.584,Z 419.048,A -85,B 0,C 180,E1 -15637.528,E2 -15637.528} C_VEL
LIN {X 0,Y 312.634,Z 419.04,A -85,B 0,C 180,E1 -15641.655,E2 -15641.655} C_VEL
LIN {X 0,Y 312.689,Z 419.032,A -85,B 0,C 180,E1 -15645.685,E2 -15645.685} C_VEL
LIN {X 0,Y 312.697,Z 419.031,A -85,B 0,C 180,E1 -15649.641,E2 -15649.641} C_VEL
LIN {X 0,Y 312.869,Z 419.013,A -85,B 0,C 180,E1 -15652.253,E2 -15652.253} C_VEL
LIN {X 0,Y 312.713,Z 419.032,A -85,B 0,C 180,E1 -15654.842,E2 -15654.842} C_VEL
LIN {X 0,Y 312.985,Z 418.996,A -85,B 0,C 180,E1 -15658.713,E2 -15658.713} C_VEL
LIN {X 0,Y 312.985,Z 418.988,A -85,B 0,C 180,E1 -15661.286,E2 -15661.286} C_VEL
LIN {X 0,Y 312.713,Z 419.028,A -85,B 0,C 180,E1 -15665.157,E2 -15665.157} C_VEL
LIN {X 0,Y 312.866,Z 419.012,A -85,B 0,C 180,E1 -15667.745,E2 -15667.745} C_VEL
LIN {X 0,Y 312.663,Z 419.036,A -85,B 0,C 180,E1 -15671.671,E2 -15671.671} C_VEL
LIN {X 0,Y 312.694,Z 419.03,A -85,B 0,C 180,E1 -15674.887,E2 -15674.887} C_VEL
LIN {X 0,Y 312.624,Z 419.04,A -85,B 0,C 180,E1 -15679.236,E2 -15679.236} C_VEL
LIN {X 0,Y 312.539,Z 419.051,A -85,B 0,C 180,E1 -15682.789,E2 -15682.789} C_VEL
LIN {X 0,Y 312.596,Z 419.047,A -85,B 0,C 180,E1 -15685.935,E2 -15685.935} C_VEL
LIN {X 0,Y 312.54,Z 419.053,A -85,B 0,C 180,E1 -15689.65,E2 -15689.65} C_VEL
LIN {X 0,Y 312.514,Z 419.058,A -85,B 0,C 180,E1 -15693.689,E2 -15693.689} C_VEL
LIN {X 0,Y 312.547,Z 419.052,A -85,B 0,C 180,E1 -15697.381,E2 -15697.381} C_VEL
LIN {X 0,Y 312.529,Z 419.052,A -85,B 0,C 180,E1 -15700.702,E2 -15700.702} C_VEL
LIN {X 0,Y 312.589,Z 419.046,A -85,B 0,C 180,E1 -15704.184,E2 -15704.184} C_VEL
LIN {X 0,Y 312.551,Z 419.053,A -85,B 0,C 180,E1 -15707.904,E2 -15707.904} C_VEL
LIN {X 0,Y 312.552,Z 419.052,A -85,B 0,C 180,E1 -15711.905,E2 -15711.905} C_VEL
LIN {X 0,Y 312.5,Z 419.06,A -85,B 0,C 180,E1 -15715.79,E2 -15715.79} C_VEL
LIN {X 0,Y 312.518,Z 419.055,A -85,B 0,C 180,E1 -15718.854,E2 -15718.854} C_VEL
LIN {X 0,Y 312.569,Z 419.05,A -85,B 0,C 180,E1 -15721.825,E2 -15721.825} C_VEL
LIN {X 0,Y 312.581,Z 419.048,A -85,B 0,C 180,E1 -15724.711,E2 -15724.711} C_VEL
LIN {X 0,Y 312.561,Z 419.207,A -85,B 0,C 180,E1 -15726.362,E2 -15726.362} C_VEL
LIN {X 0,Y 313.592,Z 422.022,A -85,B 0,C 180,E1 -15726.526,E2 -15726.526} C_VEL
LIN {X 0,Y 316.624,Z 426.927,A -85,B 0,C 180,E1 -15726.947,E2 -15726.947} C_VEL
LIN {X 0,Y 319.716,Z 431.511,A -85,B 0,C 180,E1 -15727.403,E2 -15727.403} C_VEL
LIN {X 0,Y 323.573,Z 436.682,A -85,B 0,C 180,E1 -15728.034,E2 -15728.034} C_VEL
LIN {X 0,Y 328.043,Z 442.293,A -85,B 0,C 180,E1 -15728.824,E2 -15728.824} C_VEL
LIN {X 0,Y 332.629,Z 447.74,A -85,B 0,C 180,E1 -15729.697,E2 -15729.697} C_VEL
LIN {X 0,Y 338.082,Z 453.925,A -85,B 0,C 180,E1 -15730.833,E2 -15730.833} C_VEL
LIN {X 0,Y 343.703,Z 459.958,A -85,B 0,C 180,E1 -15732.104,E2 -15732.104} C_VEL
LIN {X 0,Y 349.937,Z 466.342,A -85,B 0,C 180,E1 -15733.67,E2 -15733.67} C_VEL
LIN {X 0,Y 353.891,Z 470.042,A -85,B 0,C 180,E1 -15734.745,E2 -15734.745} C_VEL
LIN {X 0,Y 358.296,Z 474.294,A -85,B 0,C 180,E1 -15736.084,E2 -15736.084} C_VEL
LIN {X 0,Y 361.489,Z 477.016,A -85,B 0,C 180,E1 -15737.11,E2 -15737.11} C_VEL
LIN {X 0,Y 365.586,Z 480.896,A -85,B 0,C 180,E1 -15738.639,E2 -15738.639} C_VEL
LIN {X 0,Y 369.444,Z 483.472,A -85,B 0,C 180,E1 -15740.142,E2 -15740.142} C_VEL
LIN {X 0,Y 371.646,Z 485.821,A -85,B 0,C 180,E1 -15741.299,E2 -15741.299} C_VEL
LIN {X 0,Y 373.543,Z 487.761,A -85,B 0,C 180,E1 -15742.432,E2 -15742.432} C_VEL
LIN {X 0,Y 375.324,Z 489.153,A -85,B 0,C 180,E1 -15743.549,E2 -15743.549} C_VEL
LIN {X 0,Y 376.832,Z 490.147,A -85,B 0,C 180,E1 -15744.65,E2 -15744.65} C_VEL
LIN {X 0,Y 378.137,Z 490.769,A -85,B 0,C 180,E1 -15745.737,E2 -15745.737} C_VEL
LIN {X 0,Y 379.84,Z 491.2,A -85,B 0,C 180,E1 -15747.599,E2 -15747.599} C_VEL
LIN {X 0,Y 380.536,Z 491.297,A -85,B 0,C 180,E1 -15748.942,E2 -15748.942} C_VEL
LIN {X 0,Y 380.672,Z 491.37,A -85,B 0,C 180,E1 -15750,E2 -15750} C_VEL
LIN {X 0,Y 380.525,Z 491.291,A -85,B 0,C 180,E1 -15751.058,E2 -15751.058} C_VEL
LIN {X 0,Y 379.839,Z 491.212,A -85,B 0,C 180,E1 -15752.394,E2 -15752.394} C_VEL
LIN {X 0,Y 378.164,Z 490.746,A -85,B 0,C 180,E1 -15754.263,E2 -15754.263} C_VEL
LIN {X 0,Y 376.836,Z 490.174,A -85,B 0,C 180,E1 -15755.351,E2 -15755.351} C_VEL
LIN {X 0,Y 375.005,Z 488.921,A -85,B 0,C 180,E1 -15756.654,E2 -15756.654} C_VEL
LIN {X 0,Y 373.554,Z 487.787,A -85,B 0,C 180,E1 -15757.568,E2 -15757.568} C_VEL
LIN {X 0,Y 370.39,Z 484.46,A -85,B 0,C 180,E1 -15759.367,E2 -15759.367} C_VEL
LIN {X 0,Y 369.431,Z 483.507,A -85,B 0,C 180,E1 -15759.859,E2 -15759.859} C_VEL
LIN {X 0,Y 365.579,Z 480.886,A -85,B 0,C 180,E1 -15761.355,E2 -15761.355} C_VEL
LIN {X 0,Y 363.137,Z 478.699,A -85,B 0,C 180,E1 -15762.292,E2 -15762.292} C_VEL
LIN {X 0,Y 359.528,Z 475.144,A -85,B 0,C 180,E1 -15763.567,E2 -15763.567} C_VEL
LIN {X 0,Y 355.012,Z 471.275,A -85,B 0,C 180,E1 -15764.913,E2 -15764.913} C_VEL
LIN {X 0,Y 351.023,Z 467.239,A -85,B 0,C 180,E1 -15766.051,E2 -15766.051} C_VEL
LIN {X 0,Y 346.525,Z 462.872,A -85,B 0,C 180,E1 -15767.205,E2 -15767.205} C_VEL
LIN {X 0,Y 340.27,Z 456.372,A -85,B 0,C 180,E1 -15768.68,E2 -15768.68} C_VEL
LIN {X 0,Y 333.95,Z 449.266,A -85,B 0,C 180,E1 -15770.036,E2 -15770.036} C_VEL
LIN {X 0,Y 328.78,Z 443.197,A -85,B 0,C 180,E1 -15771.036,E2 -15771.036} C_VEL
LIN {X 0,Y 324.332,Z 437.671,A -85,B 0,C 180,E1 -15771.836,E2 -15771.836} C_VEL
LIN {X 0,Y 320.438,Z 432.527,A -85,B 0,C 180,E1 -15772.481,E2 -15772.481} C_VEL
LIN {X 0,Y 317.066,Z 427.615,A -85,B 0,C 180,E1 -15772.99,E2 -15772.99} C_VEL
LIN {X 0,Y 314.605,Z 423.686,A -85,B 0,C 180,E1 -15773.341,E2 -15773.341} C_VEL
LIN {X 0,Y 312.741,Z 420.074,A -85,B 0,C 180,E1 -15773.599,E2 -15773.599} C_VEL
LIN {X 0,Y 312.535,Z 419.053,A -85,B 0,C 180,E1 -15773.667,E2 -15773.667} C_VEL
LIN {X 0,Y 312.579,Z 419.051,A -85,B 0,C 180,E1 -15776.723,E2 -15776.723} C_VEL
LIN {X 0,Y 312.541,Z 419.052,A -85,B 0,C 180,E1 -15779.65,E2 -15779.65} C_VEL
LIN {X 0,Y 312.515,Z 419.055,A -85,B 0,C 180,E1 -15783.689,E2 -15783.689} C_VEL
LIN {X 0,Y 312.548,Z 419.05,A -85,B 0,C 180,E1 -15787.382,E2 -15787.382} C_VEL
LIN {X 0,Y 312.529,Z 419.055,A -85,B 0,C 180,E1 -15790.703,E2 -15790.703} C_VEL
LIN {X 0,Y 312.529,Z 419.057,A -85,B 0,C 180,E1 -15794.195,E2 -15794.195} C_VEL
LIN {X 0,Y 312.483,Z 419.06,A -85,B 0,C 180,E1 -15797.918,E2 -15797.918} C_VEL
LIN {X 0,Y 312.531,Z 419.055,A -85,B 0,C 180,E1 -15801.911,E2 -15801.911} C_VEL
LIN {X 0,Y 312.503,Z 419.058,A -85,B 0,C 180,E1 -15805.79,E2 -15805.79} C_VEL
LIN {X 0,Y 312.524,Z 419.053,A -85,B 0,C 180,E1 -15808.855,E2 -15808.855} C_VEL
LIN {X 0,Y 312.571,Z 419.05,A -85,B 0,C 180,E1 -15811.825,E2 -15811.825} C_VEL
LIN {X 0,Y 312.582,Z 419.044,A -85,B 0,C 180,E1 -15814.711,E2 -15814.711} C_VEL
LIN {X 0,Y 312.584,Z 419.047,A -85,B 0,C 180,E1 -15817.53,E2 -15817.53} C_VEL
LIN {X 0,Y 312.635,Z 419.042,A -85,B 0,C 180,E1 -15821.657,E2 -15821.657} C_VEL
LIN {X 0,Y 312.69,Z 419.034,A -85,B 0,C 180,E1 -15825.687,E2 -15825.687} C_VEL
LIN {X 0,Y 312.699,Z 419.035,A -85,B 0,C 180,E1 -15829.643,E2 -15829.643} C_VEL
LIN {X 0,Y 312.869,Z 419.011,A -85,B 0,C 180,E1 -15832.255,E2 -15832.255} C_VEL
LIN {X 0,Y 312.715,Z 419.028,A -85,B 0,C 180,E1 -15834.843,E2 -15834.843} C_VEL
LIN {X 0,Y 312.719,Z 419.024,A -85,B 0,C 180,E1 -15836.333,E2 -15836.333} C_VEL
LIN {X 0,Y 312.188,Z 419.092,A -85,B 0,C 180,E1 -15837.411,E2 -15837.411} C_VEL
LIN {X 0,Y 309.455,Z 419.429,A -85,B 0,C 180,E1 -15839.169,E2 -15839.169} C_VEL
LIN {X 0,Y 307.05,Z 419.732,A -85,B 0,C 180,E1 -15840.594,E2 -15840.594} C_VEL
LIN {X 0,Y 305.991,Z 419.871,A -85,B 0,C 180,E1 -15841.697,E2 -15841.697} C_VEL
LIN {X 0,Y 305.895,Z 419.876,A -85,B 0,C 180,E1 -15842.07,E2 -15842.07} C_VEL
LIN {X 0,Y 305.851,Z 419.884,A -85,B 0,C 180,E1 -15846.598,E2 -15846.598} C_VEL
LIN {X 0,Y 305.734,Z 419.902,A -85,B 0,C 180,E1 -15849.26,E2 -15849.26} C_VEL
LIN {X 0,Y 305.587,Z 419.922,A -85,B 0,C 180,E1 -15853.297,E2 -15853.297} C_VEL
LIN {X 0,Y 305.593,Z 419.917,A -85,B 0,C 180,E1 -15856.021,E2 -15856.021} C_VEL
LIN {X 0,Y 305.576,Z 419.923,A -85,B 0,C 180,E1 -15859.446,E2 -15859.446} C_VEL
LIN {X 0,Y 305.49,Z 419.933,A -85,B 0,C 180,E1 -15863.042,E2 -15863.042} C_VEL
LIN {X 0,Y 305.525,Z 419.925,A -85,B 0,C 180,E1 -15866.219,E2 -15866.219} C_VEL
LIN {X 0,Y 305.488,Z 419.935,A -85,B 0,C 180,E1 -15869.048,E2 -15869.048} C_VEL
LIN {X 0,Y 305.473,Z 419.937,A -85,B 0,C 180,E1 -15873.517,E2 -15873.517} C_VEL
LIN {X 0,Y 305.758,Z 421.878,A -85,B 0,C 180,E1 -15876.701,E2 -15876.701} C_VEL
LIN {X 0,Y 306.178,Z 424.687,A -85,B 0,C 180,E1 -15880.758,E2 -15880.758} C_VEL
LIN {X 0,Y 306.53,Z 427.709,A -85,B 0,C 180,E1 -15884.704,E2 -15884.704} C_VEL
LIN {X 0,Y 306.695,Z 429.746,A -85,B 0,C 180,E1 -15887.164,E2 -15887.164} C_VEL
LIN {X 0,Y 306.509,Z 432.329,A -85,B 0,C 180,E1 -15890.058,E2 -15890.058} C_VEL
LIN {X 0,Y 306.015,Z 435.608,A -85,B 0,C 180,E1 -15893.497,E2 -15893.497} C_VEL
LIN {X 0,Y 305.548,Z 438.612,A -85,B 0,C 180,E1 -15896.494,E2 -15896.494} C_VEL
LIN {X 0,Y 305.063,Z 441.797,A -85,B 0,C 180,E1 -15899.547,E2 -15899.547} C_VEL
LIN {X 0,Y 304.696,Z 445.025,A -85,B 0,C 180,E1 -15902.528,E2 -15902.528} C_VEL
LIN {X 0,Y 304.308,Z 448.822,A -85,B 0,C 180,E1 -15906.006,E2 -15906.006} C_VEL
LIN {X 0,Y 307.148,Z 460.465,A -85,B 0,C 180,E1 -15906.758,E2 -15906.758} C_VEL
LIN {X 0,Y 309.31,Z 470.97,A -85,B 0,C 180,E1 -15907.582,E2 -15907.582} C_VEL
LIN {X 0,Y 311.147,Z 484.153,A -85,B 0,C 180,E1 -15908.814,E2 -15908.814} C_VEL
LIN {X 0,Y 311.917,Z 493.776,A -85,B 0,C 180,E1 -15909.903,E2 -15909.903} C_VEL
LIN {X 0,Y 310.467,Z 504.074,A -85,B 0,C 180,E1 -15911.181,E2 -15911.181} C_VEL
LIN {X 0,Y 309.201,Z 512.607,A -85,B 0,C 180,E1 -15912.472,E2 -15912.472} C_VEL
LIN {X 0,Y 308.099,Z 520.203,A -85,B 0,C 180,E1 -15913.851,E2 -15913.851} C_VEL
LIN {X 0,Y 306.919,Z 527.411,A -85,B 0,C 180,E1 -15915.411,E2 -15915.411} C_VEL
LIN {X 0,Y 305.836,Z 533.729,A -85,B 0,C 180,E1 -15917.053,E2 -15917.053} C_VEL
LIN {X 0,Y 305.067,Z 538.995,A -85,B 0,C 180,E1 -15918.707,E2 -15918.707} C_VEL
LIN {X 0,Y 304.347,Z 544.128,A -85,B 0,C 180,E1 -15920.697,E2 -15920.697} C_VEL
LIN {X 0,Y 303.876,Z 548.12,A -85,B 0,C 180,E1 -15922.692,E2 -15922.692} C_VEL
LIN {X 0,Y 303.688,Z 551.074,A -85,B 0,C 180,E1 -15924.688,E2 -15924.688} C_VEL
LIN {X 0,Y 303.609,Z 553.525,A -85,B 0,C 180,E1 -15927.346,E2 -15927.346} C_VEL
LIN {X 0,Y 303.561,Z 554.114,A -85,B 0,C 180,E1 -15928.673,E2 -15928.673} C_VEL
LIN {X 0,Y 303.561,Z 554.115,A -85,B 0,C 180,E1 -15931.326,E2 -15931.326} C_VEL
LIN {X 0,Y 303.609,Z 553.526,A -85,B 0,C 180,E1 -15932.653,E2 -15932.653} C_VEL
LIN {X 0,Y 303.688,Z 551.075,A -85,B 0,C 180,E1 -15935.311,E2 -15935.311} C_VEL
LIN {X 0,Y 303.934,Z 548.122,A -85,B 0,C 180,E1 -15937.306,E2 -15937.306} C_VEL
LIN {X 0,Y 304.346,Z 544.13,A -85,B 0,C 180,E1 -15939.302,E2 -15939.302} C_VEL
LIN {X 0,Y 305.067,Z 538.997,A -85,B 0,C 180,E1 -15941.292,E2 -15941.292} C_VEL
LIN {X 0,Y 305.836,Z 533.731,A -85,B 0,C 180,E1 -15942.947,E2 -15942.947} C_VEL
LIN {X 0,Y 306.91,Z 527.413,A -85,B 0,C 180,E1 -15944.589,E2 -15944.589} C_VEL
LIN {X 0,Y 308.09,Z 520.206,A -85,B 0,C 180,E1 -15946.148,E2 -15946.148} C_VEL
LIN {X 0,Y 309.194,Z 512.61,A -85,B 0,C 180,E1 -15947.528,E2 -15947.528} C_VEL
LIN {X 0,Y 310.452,Z 504.077,A -85,B 0,C 180,E1 -15948.819,E2 -15948.819} C_VEL
LIN {X 0,Y 311.923,Z 493.781,A -85,B 0,C 180,E1 -15950.096,E2 -15950.096} C_VEL
LIN {X 0,Y 310.812,Z 481.211,A -85,B 0,C 180,E1 -15951.477,E2 -15951.477} C_VEL
LIN {X 0,Y 309.31,Z 470.974,A -85,B 0,C 180,E1 -15952.418,E2 -15952.418} C_VEL
LIN {X 0,Y 307.085,Z 460.087,A -85,B 0,C 180,E1 -15953.267,E2 -15953.267} C_VEL
LIN {X 0,Y 304.352,Z 449.385,A -85,B 0,C 180,E1 -15953.96,E2 -15953.96} C_VEL
LIN {X 0,Y 304.289,Z 448.805,A -85,B 0,C 180,E1 -15954.01,E2 -15954.01} C_VEL
LIN {X 0,Y 304.689,Z 444.979,A -85,B 0,C 180,E1 -15957.472,E2 -15957.472} C_VEL
LIN {X 0,Y 305.227,Z 440.607,A -85,B 0,C 180,E1 -15961.575,E2 -15961.575} C_VEL
LIN {X 0,Y 305.779,Z 437.022,A -85,B 0,C 180,E1 -15965.071,E2 -15965.071} C_VEL
LIN {X 0,Y 306.354,Z 433.448,A -85,B 0,C 180,E1 -15968.74,E2 -15968.74} C_VEL
LIN {X 0,Y 306.667,Z 430.775,A -85,B 0,C 180,E1 -15971.651,E2 -15971.651} C_VEL
LIN {X 0,Y 306.578,Z 428.167,A -85,B 0,C 180,E1 -15974.712,E2 -15974.712} C_VEL
LIN {X 0,Y 306.253,Z 425.383,A -85,B 0,C 180,E1 -15978.278,E2 -15978.278} C_VEL
LIN {X 0,Y 305.878,Z 422.976,A -85,B 0,C 180,E1 -15981.656,E2 -15981.656} C_VEL
LIN {X 0,Y 305.598,Z 420.868,A -85,B 0,C 180,E1 -15984.904,E2 -15984.904} C_VEL
LIN {X 0,Y 305.473,Z 419.937,A -85,B 0,C 180,E1 -15986.483,E2 -15986.483} C_VEL
LIN {X 0,Y 305.494,Z 419.934,A -85,B 0,C 180,E1 -15990.949,E2 -15990.949} C_VEL
LIN {X 0,Y 305.568,Z 419.922,A -85,B 0,C 180,E1 -15994.087,E2 -15994.087} C_VEL
LIN {X 0,Y 305.497,Z 419.933,A -85,B 0,C 180,E1 -15998.402,E2 -15998.402} C_VEL
LIN {X 0,Y 305.586,Z 419.919,A -85,B 0,C 180,E1 -16001.217,E2 -16001.217} C_VEL
LIN {X 0,Y 305.645,Z 419.91,A -85,B 0,C 180,E1 -16005.348,E2 -16005.348} C_VEL
LIN {X 0,Y 305.634,Z 419.912,A -85,B 0,C 180,E1 -16009.399,E2 -16009.399} C_VEL
LIN {X 0,Y 305.81,Z 419.891,A -85,B 0,C 180,E1 -16012.074,E2 -16012.074} C_VEL
LIN {X 0,Y 305.685,Z 419.908,A -85,B 0,C 180,E1 -16014.723,E2 -16014.723} C_VEL
LIN {X 0,Y 305.952,Z 419.872,A -85,B 0,C 180,E1 -16018.683,E2 -16018.683} C_VEL
LIN {X 0,Y 305.952,Z 419.863,A -85,B 0,C 180,E1 -16021.316,E2 -16021.316} C_VEL
LIN {X 0,Y 305.846,Z 419.888,A -85,B 0,C 180,E1 -16026.597,E2 -16026.597} C_VEL
LIN {X 0,Y 305.73,Z 419.898,A -85,B 0,C 180,E1 -16029.259,E2 -16029.259} C_VEL
LIN {X 0,Y 305.582,Z 419.918,A -85,B 0,C 180,E1 -16033.296,E2 -16033.296} C_VEL
LIN {X 0,Y 305.588,Z 419.919,A -85,B 0,C 180,E1 -16036.02,E2 -16036.02} C_VEL
LIN {X 0,Y 305.571,Z 419.919,A -85,B 0,C 180,E1 -16039.445,E2 -16039.445} C_VEL
LIN {X 0,Y 305.484,Z 419.93,A -85,B 0,C 180,E1 -16043.041,E2 -16043.041} C_VEL
LIN {X 0,Y 305.541,Z 419.926,A -85,B 0,C 180,E1 -16046.227,E2 -16046.227} C_VEL
LIN {X 0,Y 305.49,Z 419.929,A -85,B 0,C 180,E1 -16049.05,E2 -16049.05} C_VEL
LIN {X 0,Y 305.442,Z 419.94,A -85,B 0,C 180,E1 -16051.951,E2 -16051.951} C_VEL
LIN {X 0,Y 305.457,Z 419.934,A -85,B 0,C 180,E1 -16055.113,E2 -16055.113} C_VEL
LIN {X 0,Y 305.488,Z 419.93,A -85,B 0,C 180,E1 -16058.539,E2 -16058.539} C_VEL
LIN {X 0,Y 305.515,Z 419.926,A -85,B 0,C 180,E1 -16062.599,E2 -16062.599} C_VEL
LIN {X 0,Y 305.528,Z 419.925,A -85,B 0,C 180,E1 -16066.364,E2 -16066.364} C_VEL
LIN {X 0,Y 305.494,Z 419.932,A -85,B 0,C 180,E1 -16069.899,E2 -16069.899} C_VEL
LIN {X 0,Y 305.496,Z 419.933,A -85,B 0,C 180,E1 -16073.626,E2 -16073.626} C_VEL
LIN {X 0,Y 305.459,Z 419.934,A -85,B 0,C 180,E1 -16076.483,E2 -16076.483} C_VEL
LIN {X 0,Y 305.49,Z 419.932,A -85,B 0,C 180,E1 -16080.95,E2 -16080.95} C_VEL
LIN {X 0,Y 305.567,Z 419.922,A -85,B 0,C 180,E1 -16084.088,E2 -16084.088} C_VEL
LIN {X 0,Y 305.496,Z 419.932,A -85,B 0,C 180,E1 -16085.749,E2 -16085.749} C_VEL
LIN {X 0,Y 306.525,Z 422.791,A -85,B 0,C 180,E1 -16085.922,E2 -16085.922} C_VEL
LIN {X 0,Y 310.607,Z 430.232,A -85,B 0,C 180,E1 -16086.465,E2 -16086.465} C_VEL
LIN {X 0,Y 316.507,Z 438.853,A -85,B 0,C 180,E1 -16087.35,E2 -16087.35} C_VEL
LIN {X 0,Y 323.359,Z 447.372,A -85,B 0,C 180,E1 -16088.518,E2 -16088.518} C_VEL
LIN {X 0,Y 329.645,Z 454.772,A -85,B 0,C 180,E1 -16089.728,E2 -16089.728} C_VEL
LIN {X 0,Y 335.367,Z 461.125,A -85,B 0,C 180,E1 -16090.948,E2 -16090.948} C_VEL
LIN {X 0,Y 340.811,Z 466.798,A -85,B 0,C 180,E1 -16092.203,E2 -16092.203} C_VEL
LIN {X 0,Y 345.709,Z 471.902,A -85,B 0,C 180,E1 -16093.465,E2 -16093.465} C_VEL
LIN {X 0,Y 349.887,Z 475.852,A -85,B 0,C 180,E1 -16094.609,E2 -16094.609} C_VEL
LIN {X 0,Y 354.764,Z 480.465,A -85,B 0,C 180,E1 -16096.094,E2 -16096.094} C_VEL
LIN {X 0,Y 357.263,Z 482.588,A -85,B 0,C 180,E1 -16096.899,E2 -16096.899} C_VEL
LIN {X 0,Y 359.574,Z 485,A -85,B 0,C 180,E1 -16097.756,E2 -16097.756} C_VEL
LIN {X 0,Y 362.392,Z 487.354,A -85,B 0,C 180,E1 -16098.818,E2 -16098.818} C_VEL
LIN {X 0,Y 365.564,Z 489.394,A -85,B 0,C 180,E1 -16100.037,E2 -16100.037} C_VEL
LIN {X 0,Y 369.071,Z 493.051,A -85,B 0,C 180,E1 -16101.968,E2 -16101.968} C_VEL
LIN {X 0,Y 371.468,Z 495.084,A -85,B 0,C 180,E1 -16103.482,E2 -16103.482} C_VEL
LIN {X 0,Y 373.782,Z 496.513,A -85,B 0,C 180,E1 -16105.214,E2 -16105.214} C_VEL
LIN {X 0,Y 375.455,Z 497.071,A -85,B 0,C 180,E1 -16106.781,E2 -16106.781} C_VEL
LIN {X 0,Y 376.286,Z 497.273,A -85,B 0,C 180,E1 -16107.86,E2 -16107.86} C_VEL
LIN {X 0,Y 376.816,Z 497.351,A -85,B 0,C 180,E1 -16108.932,E2 -16108.932} C_VEL
LIN {X 0,Y 376.973,Z 497.399,A -85,B 0,C 180,E1 -16110,E2 -16110} C_VEL
LIN {X 0,Y 376.807,Z 497.341,A -85,B 0,C 180,E1 -16111.069,E2 -16111.069} C_VEL
LIN {X 0,Y 376.271,Z 497.27,A -85,B 0,C 180,E1 -16112.141,E2 -16112.141} C_VEL
LIN {X 0,Y 375.451,Z 497.056,A -85,B 0,C 180,E1 -16113.219,E2 -16113.219} C_VEL
LIN {X 0,Y 373.779,Z 496.503,A -85,B 0,C 180,E1 -16114.781,E2 -16114.781} C_VEL
LIN {X 0,Y 371.433,Z 495.101,A -85,B 0,C 180,E1 -16116.519,E2 -16116.519} C_VEL
LIN {X 0,Y 369.067,Z 493.085,A -85,B 0,C 180,E1 -16118.027,E2 -16118.027} C_VEL
LIN {X 0,Y 365.535,Z 489.439,A -85,B 0,C 180,E1 -16119.965,E2 -16119.965} C_VEL
LIN {X 0,Y 361.463,Z 486.59,A -85,B 0,C 180,E1 -16121.539,E2 -16121.539} C_VEL
LIN {X 0,Y 357.403,Z 482.729,A -85,B 0,C 180,E1 -16123.048,E2 -16123.048} C_VEL
LIN {X 0,Y 352.817,Z 478.782,A -85,B 0,C 180,E1 -16124.499,E2 -16124.499} C_VEL
LIN {X 0,Y 346.902,Z 472.909,A -85,B 0,C 180,E1 -16126.237,E2 -16126.237} C_VEL
LIN {X 0,Y 341.874,Z 467.884,A -85,B 0,C 180,E1 -16127.535,E2 -16127.535} C_VEL
LIN {X 0,Y 336.794,Z 462.782,A -85,B 0,C 180,E1 -16128.725,E2 -16128.725} C_VEL
LIN {X 0,Y 329.645,Z 454.767,A -85,B 0,C 180,E1 -16130.272,E2 -16130.272} C_VEL
LIN {X 0,Y 324.07,Z 448.201,A -85,B 0,C 180,E1 -16131.348,E2 -16131.348} C_VEL
LIN {X 0,Y 319.48,Z 442.494,A -85,B 0,C 180,E1 -16132.171,E2 -16132.171} C_VEL
LIN {X 0,Y 315.477,Z 437.273,A -85,B 0,C 180,E1 -16132.822,E2 -16132.822} C_VEL
LIN {X 0,Y 310.243,Z 429.709,A -85,B 0,C 180,E1 -16133.583,E2 -16133.583} C_VEL
LIN {X 0,Y 307.046,Z 423.847,A -85,B 0,C 180,E1 -16134.007,E2 -16134.007} C_VEL
LIN {X 0,Y 305.554,Z 420.292,A -85,B 0,C 180,E1 -16134.223,E2 -16134.223} C_VEL
LIN {X 0,Y 305.492,Z 419.933,A -85,B 0,C 180,E1 -16134.268,E2 -16134.268} C_VEL
LIN {X 0,Y 305.53,Z 419.926,A -85,B 0,C 180,E1 -16137.39,E2 -16137.39} C_VEL
LIN {X 0,Y 305.46,Z 419.938,A -85,B 0,C 180,E1 -16140.409,E2 -16140.409} C_VEL
LIN {X 0,Y 305.46,Z 419.936,A -85,B 0,C 180,E1 -16144.079,E2 -16144.079} C_VEL
LIN {X 0,Y 305.498,Z 419.931,A -85,B 0,C 180,E1 -16146.736,E2 -16146.736} C_VEL
LIN {X 0,Y 305.49,Z 419.933,A -85,B 0,C 180,E1 -16150.609,E2 -16150.609} C_VEL
LIN {X 0,Y 305.488,Z 419.93,A -85,B 0,C 180,E1 -16153.643,E2 -16153.643} C_VEL
LIN {X 0,Y 305.459,Z 419.933,A -85,B 0,C 180,E1 -16157.413,E2 -16157.413} C_VEL
LIN {X 0,Y 305.491,Z 419.93,A -85,B 0,C 180,E1 -16161.601,E2 -16161.601} C_VEL
LIN {X 0,Y 305.459,Z 419.934,A -85,B 0,C 180,E1 -16164.887,E2 -16164.887} C_VEL
LIN {X 0,Y 305.452,Z 419.937,A -85,B 0,C 180,E1 -16168.354,E2 -16168.354} C_VEL
LIN {X 0,Y 305.517,Z 419.925,A -85,B 0,C 180,E1 -16171.114,E2 -16171.114} C_VEL
LIN {X 0,Y 305.568,Z 419.922,A -85,B 0,C 180,E1 -16174.088,E2 -16174.088} C_VEL
LIN {X 0,Y 305.497,Z 419.929,A -85,B 0,C 180,E1 -16178.403,E2 -16178.403} C_VEL
LIN {X 0,Y 305.587,Z 419.917,A -85,B 0,C 180,E1 -16181.218,E2 -16181.218} C_VEL
LIN {X 0,Y 305.646,Z 419.909,A -85,B 0,C 180,E1 -16185.35,E2 -16185.35} C_VEL
LIN {X 0,Y 305.635,Z 419.913,A -85,B 0,C 180,E1 -16189.4,E2 -16189.4} C_VEL
LIN {X 0,Y 305.81,Z 419.892,A -85,B 0,C 180,E1 -16192.075,E2 -16192.075} C_VEL
LIN {X 0,Y 305.687,Z 419.903,A -85,B 0,C 180,E1 -16194.724,E2 -16194.724} C_VEL
LIN {X 0,Y 305.955,Z 419.863,A -85,B 0,C 180,E1 -16198.684,E2 -16198.684} C_VEL
LIN {X 0,Y 305.955,Z 419.872,A -85,B 0,C 180,E1 -16201.317,E2 -16201.317} C_VEL
LIN {X 0,Y 305.895,Z 419.876,A -85,B 0,C 180,E1 -16202.07,E2 -16202.07} C_VEL
LIN {X 0,Y 305.19,Z 419.97,A -85,B 0,C 180,E1 -16203.167,E2 -16203.167} C_VEL
LIN {X 0,Y 302.29,Z 420.329,A -85,B 0,C 180,E1 -16204.952,E2 -16204.952} C_VEL
LIN {X 0,Y 299.858,Z 420.631,A -85,B 0,C 180,E1 -16206.401,E2 -16206.401} C_VEL
LIN {X 0,Y 298.83,Z 420.764,A -85,B 0,C 180,E1 -16207.523,E2 -16207.523} C_VEL
LIN {X 0,Y 298.753,Z 420.768,A -85,B 0,C 180,E1 -16207.903,E2 -16207.903} C_VEL
LIN {X 0,Y 298.592,Z 420.79,A -85,B 0,C 180,E1 -16210.854,E2 -16210.854} C_VEL
LIN {X 0,Y 298.605,Z 420.791,A -85,B 0,C 180,E1 -16215.21,E2 -16215.21} C_VEL
LIN {X 0,Y 298.539,Z 420.8,A -85,B 0,C 180,E1 -16219.244,E2 -16219.244} C_VEL
LIN {X 0,Y 298.457,Z 420.809,A -85,B 0,C 180,E1 -16223.598,E2 -16223.598} C_VEL
LIN {X 0,Y 298.485,Z 420.803,A -85,B 0,C 180,E1 -16226.576,E2 -16226.576} C_VEL
LIN {X 0,Y 298.416,Z 420.816,A -85,B 0,C 180,E1 -16229.642,E2 -16229.642} C_VEL
LIN {X 0,Y 298.399,Z 420.818,A -85,B 0,C 180,E1 -16232.801,E2 -16232.801} C_VEL
LIN {X 0,Y 298.673,Z 422.561,A -85,B 0,C 180,E1 -16236.035,E2 -16236.035} C_VEL
LIN {X 0,Y 298.972,Z 424.781,A -85,B 0,C 180,E1 -16239.398,E2 -16239.398} C_VEL
LIN {X 0,Y 299.347,Z 427.313,A -85,B 0,C 180,E1 -16242.911,E2 -16242.911} C_VEL
LIN {X 0,Y 299.656,Z 430.244,A -85,B 0,C 180,E1 -16246.641,E2 -16246.641} C_VEL
LIN {X 0,Y 299.577,Z 432.212,A -85,B 0,C 180,E1 -16248.938,E2 -16248.938} C_VEL
LIN {X 0,Y 299.111,Z 435.318,A -85,B 0,C 180,E1 -16252.345,E2 -16252.345} C_VEL
LIN {X 0,Y 298.644,Z 438.467,A -85,B 0,C 180,E1 -16255.612,E2 -16255.612} C_VEL
LIN {X 0,Y 298.108,Z 441.637,A -85,B 0,C 180,E1 -16258.758,E2 -16258.758} C_VEL
LIN {X 0,Y 297.685,Z 444.825,A -85,B 0,C 180,E1 -16261.824,E2 -16261.824} C_VEL
LIN {X 0,Y 297.272,Z 448.701,A -85,B 0,C 180,E1 -16265.417,E2 -16265.417} C_VEL
LIN {X 0,Y 299.74,Z 458.329,A -85,B 0,C 180,E1 -16266.049,E2 -16266.049} C_VEL
LIN {X 0,Y 301.957,Z 468.318,A -85,B 0,C 180,E1 -16266.835,E2 -16266.835} C_VEL
LIN {X 0,Y 303.315,Z 476.954,A -85,B 0,C 180,E1 -16267.608,E2 -16267.608} C_VEL
LIN {X 0,Y 304.414,Z 485.579,A -85,B 0,C 180,E1 -16268.5,E2 -16268.5} C_VEL
LIN {X 0,Y 305.057,Z 494.916,A -85,B 0,C 180,E1 -16269.607,E2 -16269.607} C_VEL
LIN {X 0,Y 303.723,Z 503.862,A -85,B 0,C 180,E1 -16270.747,E2 -16270.747} C_VEL
LIN {X 0,Y 302.406,Z 512.394,A -85,B 0,C 180,E1 -16272.065,E2 -16272.065} C_VEL
LIN {X 0,Y 301.243,Z 520.156,A -85,B 0,C 180,E1 -16273.509,E2 -16273.509} C_VEL
LIN {X 0,Y 300.019,Z 527.199,A -85,B 0,C 180,E1 -16275.068,E2 -16275.068} C_VEL
LIN {X 0,Y 298.903,Z 533.517,A -85,B 0,C 180,E1 -16276.747,E2 -16276.747} C_VEL
LIN {X 0,Y 298.082,Z 538.783,A -85,B 0,C 180,E1 -16278.439,E2 -16278.439} C_VEL
LIN {X 0,Y 297.313,Z 543.916,A -85,B 0,C 180,E1 -16280.475,E2 -16280.475} C_VEL
LIN {X 0,Y 296.822,Z 547.908,A -85,B 0,C 180,E1 -16282.517,E2 -16282.517} C_VEL
LIN {X 0,Y 296.603,Z 550.862,A -85,B 0,C 180,E1 -16284.561,E2 -16284.561} C_VEL
LIN {X 0,Y 296.536,Z 553.315,A -85,B 0,C 180,E1 -16287.283,E2 -16287.283} C_VEL
LIN {X 0,Y 296.481,Z 553.904,A -85,B 0,C 180,E1 -16288.641,E2 -16288.641} C_VEL
LIN {X 0,Y 296.481,Z 553.904,A -85,B 0,C 180,E1 -16291.358,E2 -16291.358} C_VEL
LIN {X 0,Y 296.536,Z 553.315,A -85,B 0,C 180,E1 -16292.717,E2 -16292.717} C_VEL
LIN {X 0,Y 296.603,Z 550.863,A -85,B 0,C 180,E1 -16295.438,E2 -16295.438} C_VEL
LIN {X 0,Y 296.858,Z 547.91,A -85,B 0,C 180,E1 -16297.481,E2 -16297.481} C_VEL
LIN {X 0,Y 297.313,Z 543.917,A -85,B 0,C 180,E1 -16299.524,E2 -16299.524} C_VEL
LIN {X 0,Y 298.081,Z 538.785,A -85,B 0,C 180,E1 -16301.56,E2 -16301.56} C_VEL
LIN {X 0,Y 298.903,Z 533.519,A -85,B 0,C 180,E1 -16303.252,E2 -16303.252} C_VEL
LIN {X 0,Y 300.008,Z 527.201,A -85,B 0,C 180,E1 -16304.932,E2 -16304.932} C_VEL
LIN {X 0,Y 301.236,Z 520.159,A -85,B 0,C 180,E1 -16306.491,E2 -16306.491} C_VEL
LIN {X 0,Y 302.403,Z 512.397,A -85,B 0,C 180,E1 -16307.934,E2 -16307.934} C_VEL
LIN {X 0,Y 303.707,Z 503.865,A -85,B 0,C 180,E1 -16309.253,E2 -16309.253} C_VEL
LIN {X 0,Y 305.125,Z 493.565,A -85,B 0,C 180,E1 -16310.564,E2 -16310.564} C_VEL
LIN {X 0,Y 304.086,Z 482.364,A -85,B 0,C 180,E1 -16311.856,E2 -16311.856} C_VEL
LIN {X 0,Y 302.421,Z 470.912,A -85,B 0,C 180,E1 -16312.946,E2 -16312.946} C_VEL
LIN {X 0,Y 300.054,Z 459.706,A -85,B 0,C 180,E1 -16313.853,E2 -16313.853} C_VEL
LIN {X 0,Y 297.342,Z 449.3,A -85,B 0,C 180,E1 -16314.556,E2 -16314.556} C_VEL
LIN {X 0,Y 297.265,Z 448.62,A -85,B 0,C 180,E1 -16314.604,E2 -16314.604} C_VEL
LIN {X 0,Y 297.68,Z 444.809,A -85,B 0,C 180,E1 -16318.175,E2 -16318.175} C_VEL
LIN {X 0,Y 298.198,Z 440.894,A -85,B 0,C 180,E1 -16321.955,E2 -16321.955} C_VEL
LIN {X 0,Y 298.862,Z 436.885,A -85,B 0,C 180,E1 -16326.007,E2 -16326.007} C_VEL
LIN {X 0,Y 299.375,Z 433.758,A -85,B 0,C 180,E1 -16329.333,E2 -16329.333} C_VEL
LIN {X 0,Y 299.671,Z 430.652,A -85,B 0,C 180,E1 -16332.852,E2 -16332.852} C_VEL
LIN {X 0,Y 299.391,Z 427.596,A -85,B 0,C 180,E1 -16336.693,E2 -16336.693} C_VEL
LIN {X 0,Y 298.962,Z 424.762,A -85,B 0,C 180,E1 -16340.6,E2 -16340.6} C_VEL
LIN {X 0,Y 298.673,Z 422.563,A -85,B 0,C 180,E1 -16343.965,E2 -16343.965} C_VEL
LIN {X 0,Y 298.4,Z 420.819,A -85,B 0,C 180,E1 -16347.2,E2 -16347.2} C_VEL
LIN {X 0,Y 298.43,Z 420.813,A -85,B 0,C 180,E1 -16350.613,E2 -16350.613} C_VEL
LIN {X 0,Y 298.481,Z 420.806,A -85,B 0,C 180,E1 -16353.473,E2 -16353.473} C_VEL
LIN {X 0,Y 298.432,Z 420.816,A -85,B 0,C 180,E1 -16356.696,E2 -16356.696} C_VEL
LIN {X 0,Y 298.536,Z 420.801,A -85,B 0,C 180,E1 -16360.756,E2 -16360.756} C_VEL
LIN {X 0,Y 298.589,Z 420.791,A -85,B 0,C 180,E1 -16364.994,E2 -16364.994} C_VEL
LIN {X 0,Y 298.589,Z 420.79,A -85,B 0,C 180,E1 -16369.146,E2 -16369.146} C_VEL
LIN {X 0,Y 298.755,Z 420.769,A -85,B 0,C 180,E1 -16371.885,E2 -16371.885} C_VEL
LIN {X 0,Y 298.656,Z 420.785,A -85,B 0,C 180,E1 -16374.598,E2 -16374.598} C_VEL
LIN {X 0,Y 298.918,Z 420.748,A -85,B 0,C 180,E1 -16378.652,E2 -16378.652} C_VEL
LIN {X 0,Y 298.918,Z 420.739,A -85,B 0,C 180,E1 -16381.346,E2 -16381.346} C_VEL
LIN {X 0,Y 298.792,Z 420.765,A -85,B 0,C 180,E1 -16386.753,E2 -16386.753} C_VEL
LIN {X 0,Y 298.675,Z 420.777,A -85,B 0,C 180,E1 -16389.48,E2 -16389.48} C_VEL
LIN {X 0,Y 298.546,Z 420.795,A -85,B 0,C 180,E1 -16393.615,E2 -16393.615} C_VEL
LIN {X 0,Y 298.543,Z 420.798,A -85,B 0,C 180,E1 -16396.408,E2 -16396.408} C_VEL
LIN {X 0,Y 298.505,Z 420.8,A -85,B 0,C 180,E1 -16399.654,E2 -16399.654} C_VEL
LIN {X 0,Y 298.451,Z 420.808,A -85,B 0,C 180,E1 -16403.597,E2 -16403.597} C_VEL
LIN {X 0,Y 298.483,Z 420.803,A -85,B 0,C 180,E1 -16406.574,E2 -16406.574} C_VEL
LIN {X 0,Y 298.416,Z 420.813,A -85,B 0,C 180,E1 -16409.641,E2 -16409.641} C_VEL
LIN {X 0,Y 298.391,Z 420.814,A -85,B 0,C 180,E1 -16412.8,E2 -16412.8} C_VEL
LIN {X 0,Y 298.464,Z 420.805,A -85,B 0,C 180,E1 -16416.814,E2 -16416.814} C_VEL
LIN {X 0,Y 298.45,Z 420.807,A -85,B 0,C 180,E1 -16421.249,E2 -16421.249} C_VEL
LIN {X 0,Y 298.483,Z 420.803,A -85,B 0,C 180,E1 -16425.061,E2 -16425.061} C_VEL
LIN {X 0,Y 298.451,Z 420.807,A -85,B 0,C 180,E1 -16428.897,E2 -16428.897} C_VEL
LIN {X 0,Y 298.464,Z 420.807,A -85,B 0,C 180,E1 -16433.186,E2 -16433.186} C_VEL
LIN {X 0,Y 298.39,Z 420.817,A -85,B 0,C 180,E1 -16437.2,E2 -16437.2} C_VEL
LIN {X 0,Y 298.464,Z 420.807,A -85,B 0,C 180,E1 -16441.905,E2 -16441.905} C_VEL
LIN {X 0,Y 298.464,Z 420.809,A -85,B 0,C 180,E1 -16445.156,E2 -16445.156} C_VEL
LIN {X 0,Y 299.496,Z 423.718,A -85,B 0,C 180,E1 -16445.338,E2 -16445.338} C_VEL
LIN {X 0,Y 304.322,Z 433.161,A -85,B 0,C 180,E1 -16446.033,E2 -16446.033} C_VEL
LIN {X 0,Y 309.642,Z 440.949,A -85,B 0,C 180,E1 -16446.813,E2 -16446.813} C_VEL
LIN {X 0,Y 313.85,Z 446.603,A -85,B 0,C 180,E1 -16447.492,E2 -16447.492} C_VEL
LIN {X 0,Y 320.386,Z 454.8,A -85,B 0,C 180,E1 -16448.664,E2 -16448.664} C_VEL
LIN {X 0,Y 327.149,Z 462.646,A -85,B 0,C 180,E1 -16450.026,E2 -16450.026} C_VEL
LIN {X 0,Y 333.585,Z 469.579,A -85,B 0,C 180,E1 -16451.45,E2 -16451.45} C_VEL
LIN {X 0,Y 339.678,Z 475.808,A -85,B 0,C 180,E1 -16452.94,E2 -16452.94} C_VEL
LIN {X 0,Y 345.082,Z 480.926,A -85,B 0,C 180,E1 -16454.389,E2 -16454.389} C_VEL
LIN {X 0,Y 348.524,Z 484.415,A -85,B 0,C 180,E1 -16455.445,E2 -16455.445} C_VEL
LIN {X 0,Y 353.396,Z 488.715,A -85,B 0,C 180,E1 -16457.02,E2 -16457.02} C_VEL
LIN {X 0,Y 358.197,Z 493.071,A -85,B 0,C 180,E1 -16458.816,E2 -16458.816} C_VEL
LIN {X 0,Y 361.101,Z 494.927,A -85,B 0,C 180,E1 -16459.912,E2 -16459.912} C_VEL
LIN {X 0,Y 363.344,Z 497.237,A -85,B 0,C 180,E1 -16461.099,E2 -16461.099} C_VEL
LIN {X 0,Y 365.277,Z 499.219,A -85,B 0,C 180,E1 -16462.26,E2 -16462.26} C_VEL
LIN {X 0,Y 367.612,Z 501.023,A -85,B 0,C 180,E1 -16463.784,E2 -16463.784} C_VEL
LIN {X 0,Y 370.002,Z 502.395,A -85,B 0,C 180,E1 -16465.643,E2 -16465.643} C_VEL
LIN {X 0,Y 371.195,Z 502.773,A -85,B 0,C 180,E1 -16466.744,E2 -16466.744} C_VEL
LIN {X 0,Y 372.071,Z 503.008,A -85,B 0,C 180,E1 -16467.835,E2 -16467.835} C_VEL
LIN {X 0,Y 372.642,Z 503.093,A -85,B 0,C 180,E1 -16468.92,E2 -16468.92} C_VEL
LIN {X 0,Y 372.806,Z 503.147,A -85,B 0,C 180,E1 -16470,E2 -16470} C_VEL
LIN {X 0,Y 372.565,Z 503.071,A -85,B 0,C 180,E1 -16471.23,E2 -16471.23} C_VEL
LIN {X 0,Y 371.188,Z 502.76,A -85,B 0,C 180,E1 -16473.256,E2 -16473.256} C_VEL
LIN {X 0,Y 370.019,Z 502.375,A -85,B 0,C 180,E1 -16474.357,E2 -16474.357} C_VEL
LIN {X 0,Y 367.61,Z 501.055,A -85,B 0,C 180,E1 -16476.213,E2 -16476.213} C_VEL
LIN {X 0,Y 365.26,Z 499.226,A -85,B 0,C 180,E1 -16477.741,E2 -16477.741} C_VEL
LIN {X 0,Y 362.983,Z 496.86,A -85,B 0,C 180,E1 -16479.091,E2 -16479.091} C_VEL
LIN {X 0,Y 361.059,Z 494.958,A -85,B 0,C 180,E1 -16480.09,E2 -16480.09} C_VEL
LIN {X 0,Y 356.304,Z 491.46,A -85,B 0,C 180,E1 -16481.906,E2 -16481.906} C_VEL
LIN {X 0,Y 351.938,Z 487.276,A -85,B 0,C 180,E1 -16483.498,E2 -16483.498} C_VEL
LIN {X 0,Y 347.274,Z 483.222,A -85,B 0,C 180,E1 -16484.944,E2 -16484.944} C_VEL
LIN {X 0,Y 342.285,Z 478.269,A -85,B 0,C 180,E1 -16486.395,E2 -16486.395} C_VEL
LIN {X 0,Y 336.306,Z 472.255,A -85,B 0,C 180,E1 -16487.915,E2 -16487.915} C_VEL
LIN {X 0,Y 330.635,Z 466.305,A -85,B 0,C 180,E1 -16489.24,E2 -16489.24} C_VEL
LIN {X 0,Y 324.77,Z 459.767,A -85,B 0,C 180,E1 -16490.484,E2 -16490.484} C_VEL
LIN {X 0,Y 317.901,Z 451.709,A -85,B 0,C 180,E1 -16491.798,E2 -16491.798} C_VEL
LIN {X 0,Y 311.03,Z 443.018,A -85,B 0,C 180,E1 -16492.961,E2 -16492.961} C_VEL
LIN {X 0,Y 305.401,Z 434.812,A -85,B 0,C 180,E1 -16493.81,E2 -16493.81} C_VEL
LIN {X 0,Y 301.168,Z 427.158,A -85,B 0,C 180,E1 -16494.426,E2 -16494.426} C_VEL
LIN {X 0,Y 298.574,Z 421.478,A -85,B 0,C 180,E1 -16494.802,E2 -16494.802} C_VEL
LIN {X 0,Y 298.475,Z 420.807,A -85,B 0,C 180,E1 -16494.877,E2 -16494.877} C_VEL
LIN {X 0,Y 298.466,Z 420.807,A -85,B 0,C 180,E1 -16498.095,E2 -16498.095} C_VEL
LIN {X 0,Y 298.391,Z 420.817,A -85,B 0,C 180,E1 -16502.8,E2 -16502.8} C_VEL
LIN {X 0,Y 298.466,Z 420.807,A -85,B 0,C 180,E1 -16506.814,E2 -16506.814} C_VEL
LIN {X 0,Y 298.451,Z 420.807,A -85,B 0,C 180,E1 -16511.103,E2 -16511.103} C_VEL
LIN {X 0,Y 298.455,Z 420.806,A -85,B 0,C 180,E1 -16513.116,E2 -16513.116} C_VEL
LIN {X 0,Y 298.428,Z 420.809,A -85,B 0,C 180,E1 -16516.926,E2 -16516.926} C_VEL
LIN {X 0,Y 298.411,Z 420.811,A -85,B 0,C 180,E1 -16521.004,E2 -16521.004} C_VEL
LIN {X 0,Y 298.428,Z 420.812,A -85,B 0,C 180,E1 -16523.933,E2 -16523.933} C_VEL
LIN {X 0,Y 298.396,Z 420.817,A -85,B 0,C 180,E1 -16527.983,E2 -16527.983} C_VEL
LIN {X 0,Y 298.46,Z 420.809,A -85,B 0,C 180,E1 -16531.905,E2 -16531.905} C_VEL
LIN {X 0,Y 298.482,Z 420.799,A -85,B 0,C 180,E1 -16534.925,E2 -16534.925} C_VEL
LIN {X 0,Y 298.447,Z 420.806,A -85,B 0,C 180,E1 -16539.316,E2 -16539.316} C_VEL
LIN {X 0,Y 298.535,Z 420.798,A -85,B 0,C 180,E1 -16542.18,E2 -16542.18} C_VEL
LIN {X 0,Y 298.59,Z 420.786,A -85,B 0,C 180,E1 -16544.995,E2 -16544.995} C_VEL
LIN {X 0,Y 298.59,Z 420.789,A -85,B 0,C 180,E1 -16549.147,E2 -16549.147} C_VEL
LIN {X 0,Y 298.756,Z 420.772,A -85,B 0,C 180,E1 -16551.887,E2 -16551.887} C_VEL
LIN {X 0,Y 298.658,Z 420.779,A -85,B 0,C 180,E1 -16554.6,E2 -16554.6} C_VEL
LIN {X 0,Y 298.921,Z 420.738,A -85,B 0,C 180,E1 -16558.654,E2 -16558.654} C_VEL
LIN {X 0,Y 298.921,Z 420.748,A -85,B 0,C 180,E1 -16561.348,E2 -16561.348} C_VEL
LIN {X 0,Y 298.796,Z 420.763,A -85,B 0,C 180,E1 -16566.755,E2 -16566.755} C_VEL
LIN {X 0,Y 298.753,Z 420.768,A -85,B 0,C 180,E1 -16567.903,E2 -16567.903} C_VEL
LIN {X 0,Y 298.073,Z 420.857,A -85,B 0,C 180,E1 -16569.027,E2 -16569.027} C_VEL
LIN {X 0,Y 295.112,Z 421.223,A -85,B 0,C 180,E1 -16570.852,E2 -16570.852} C_VEL
LIN {X 0,Y 292.616,Z 421.534,A -85,B 0,C 180,E1 -16572.335,E2 -16572.335} C_VEL
LIN {X 0,Y 291.581,Z 421.667,A -85,B 0,C 180,E1 -16573.486,E2 -16573.486} C_VEL
LIN {X 0,Y 291.516,Z 421.671,A -85,B 0,C 180,E1 -16573.876,E2 -16573.876} C_VEL
LIN {X 0,Y 291.486,Z 421.675,A -85,B 0,C 180,E1 -16576.819,E2 -16576.819} C_VEL
LIN {X 0,Y 291.45,Z 421.68,A -85,B 0,C 180,E1 -16579.876,E2 -16579.876} C_VEL
LIN {X 0,Y 291.399,Z 421.686,A -85,B 0,C 180,E1 -16584.206,E2 -16584.206} C_VEL
LIN {X 0,Y 291.419,Z 421.687,A -85,B 0,C 180,E1 -16587.273,E2 -16587.273} C_VEL
LIN {X 0,Y 291.334,Z 421.697,A -85,B 0,C 180,E1 -16590.438,E2 -16590.438} C_VEL
LIN {X 0,Y 291.345,Z 421.697,A -85,B 0,C 180,E1 -16592.405,E2 -16592.405} C_VEL
LIN {X 0,Y 291.605,Z 423.248,A -85,B 0,C 180,E1 -16595.341,E2 -16595.341} C_VEL
LIN {X 0,Y 291.964,Z 426.003,A -85,B 0,C 180,E1 -16599.621,E2 -16599.621} C_VEL
LIN {X 0,Y 292.261,Z 427.887,A -85,B 0,C 180,E1 -16602.324,E2 -16602.324} C_VEL
LIN {X 0,Y 292.574,Z 430.765,A -85,B 0,C 180,E1 -16606.108,E2 -16606.108} C_VEL
LIN {X 0,Y 292.443,Z 433.634,A -85,B 0,C 180,E1 -16609.544,E2 -16609.544} C_VEL
LIN {X 0,Y 291.962,Z 436.743,A -85,B 0,C 180,E1 -16613.002,E2 -16613.002} C_VEL
LIN {X 0,Y 291.417,Z 439.883,A -85,B 0,C 180,E1 -16616.311,E2 -16616.311} C_VEL
LIN {X 0,Y 290.792,Z 444.01,A -85,B 0,C 180,E1 -16620.467,E2 -16620.467} C_VEL
LIN {X 0,Y 290.272,Z 448.437,A -85,B 0,C 180,E1 -16624.776,E2 -16624.776} C_VEL
LIN {X 0,Y 292.048,Z 455.37,A -85,B 0,C 180,E1 -16625.23,E2 -16625.23} C_VEL
LIN {X 0,Y 294.777,Z 466.939,A -85,B 0,C 180,E1 -16626.154,E2 -16626.154} C_VEL
LIN {X 0,Y 296.281,Z 475.461,A -85,B 0,C 180,E1 -16626.931,E2 -16626.931} C_VEL
LIN {X 0,Y 297.576,Z 485.985,A -85,B 0,C 180,E1 -16628.05,E2 -16628.05} C_VEL
LIN {X 0,Y 298.216,Z 494.711,A -85,B 0,C 180,E1 -16629.119,E2 -16629.119} C_VEL
LIN {X 0,Y 297.233,Z 502.516,A -85,B 0,C 180,E1 -16630.13,E2 -16630.13} C_VEL
LIN {X 0,Y 295.953,Z 510.262,A -85,B 0,C 180,E1 -16631.302,E2 -16631.302} C_VEL
LIN {X 0,Y 294.745,Z 517.955,A -85,B 0,C 180,E1 -16632.698,E2 -16632.698} C_VEL
LIN {X 0,Y 293.383,Z 525.61,A -85,B 0,C 180,E1 -16634.366,E2 -16634.366} C_VEL
LIN {X 0,Y 292.194,Z 532.149,A -85,B 0,C 180,E1 -16636.082,E2 -16636.082} C_VEL
LIN {X 0,Y 291.377,Z 536.652,A -85,B 0,C 180,E1 -16637.462,E2 -16637.462} C_VEL
LIN {X 0,Y 290.515,Z 542.149,A -85,B 0,C 180,E1 -16639.546,E2 -16639.546} C_VEL
LIN {X 0,Y 289.917,Z 546.478,A -85,B 0,C 180,E1 -16641.637,E2 -16641.637} C_VEL
LIN {X 0,Y 289.669,Z 548.848,A -85,B 0,C 180,E1 -16643.032,E2 -16643.032} C_VEL
LIN {X 0,Y 289.519,Z 550.651,A -85,B 0,C 180,E1 -16644.428,E2 -16644.428} C_VEL
LIN {X 0,Y 289.442,Z 553.103,A -85,B 0,C 180,E1 -16647.216,E2 -16647.216} C_VEL
LIN {X 0,Y 289.404,Z 553.693,A -85,B 0,C 180,E1 -16648.608,E2 -16648.608} C_VEL
LIN {X 0,Y 289.404,Z 553.693,A -85,B 0,C 180,E1 -16651.391,E2 -16651.391} C_VEL
LIN {X 0,Y 289.442,Z 553.104,A -85,B 0,C 180,E1 -16652.783,E2 -16652.783} C_VEL
LIN {X 0,Y 289.519,Z 550.651,A -85,B 0,C 180,E1 -16655.572,E2 -16655.572} C_VEL
LIN {X 0,Y 289.81,Z 547.698,A -85,B 0,C 180,E1 -16657.664,E2 -16657.664} C_VEL
LIN {X 0,Y 290.294,Z 543.705,A -85,B 0,C 180,E1 -16659.757,E2 -16659.757} C_VEL
LIN {X 0,Y 291.08,Z 538.572,A -85,B 0,C 180,E1 -16661.842,E2 -16661.842} C_VEL
LIN {X 0,Y 291.975,Z 533.307,A -85,B 0,C 180,E1 -16663.573,E2 -16663.573} C_VEL
LIN {X 0,Y 293.113,Z 526.988,A -85,B 0,C 180,E1 -16665.292,E2 -16665.292} C_VEL
LIN {X 0,Y 294.218,Z 521.037,A -85,B 0,C 180,E1 -16666.657,E2 -16666.657} C_VEL
LIN {X 0,Y 295.293,Z 514.105,A -85,B 0,C 180,E1 -16668.023,E2 -16668.023} C_VEL
LIN {X 0,Y 296.649,Z 505.924,A -85,B 0,C 180,E1 -16669.37,E2 -16669.37} C_VEL
LIN {X 0,Y 298,Z 497.413,A -85,B 0,C 180,E1 -16670.536,E2 -16670.536} C_VEL
LIN {X 0,Y 298.228,Z 493.368,A -85,B 0,C 180,E1 -16671.058,E2 -16671.058} C_VEL
LIN {X 0,Y 297.166,Z 481.982,A -85,B 0,C 180,E1 -16672.407,E2 -16672.407} C_VEL
LIN {X 0,Y 295.532,Z 470.868,A -85,B 0,C 180,E1 -16673.5,E2 -16673.5} C_VEL
LIN {X 0,Y 293.162,Z 459.685,A -85,B 0,C 180,E1 -16674.439,E2 -16674.439} C_VEL
LIN {X 0,Y 290.306,Z 448.964,A -85,B 0,C 180,E1 -16675.196,E2 -16675.196} C_VEL
LIN {X 0,Y 290.264,Z 448.438,A -85,B 0,C 180,E1 -16675.224,E2 -16675.224} C_VEL
LIN {X 0,Y 290.787,Z 443.995,A -85,B 0,C 180,E1 -16679.531,E2 -16679.531} C_VEL
LIN {X 0,Y 291.388,Z 439.877,A -85,B 0,C 180,E1 -16683.692,E2 -16683.692} C_VEL
LIN {X 0,Y 292.009,Z 436.355,A -85,B 0,C 180,E1 -16687.416,E2 -16687.416} C_VEL
LIN {X 0,Y 292.439,Z 433.62,A -85,B 0,C 180,E1 -16690.456,E2 -16690.456} C_VEL
LIN {X 0,Y 292.573,Z 430.738,A -85,B 0,C 180,E1 -16693.892,E2 -16693.892} C_VEL
LIN {X 0,Y 292.247,Z 427.878,A -85,B 0,C 180,E1 -16697.673,E2 -16697.673} C_VEL
LIN {X 0,Y 291.864,Z 425.412,A -85,B 0,C 180,E1 -16701.238,E2 -16701.238} C_VEL
LIN {X 0,Y 291.577,Z 423.027,A -85,B 0,C 180,E1 -16705.035,E2 -16705.035} C_VEL
LIN {X 0,Y 291.374,Z 421.691,A -85,B 0,C 180,E1 -16707.95,E2 -16707.95} C_VEL
LIN {X 0,Y 291.381,Z 421.691,A -85,B 0,C 180,E1 -16711.157,E2 -16711.157} C_VEL
LIN {X 0,Y 291.414,Z 421.687,A -85,B 0,C 180,E1 -16714.271,E2 -16714.271} C_VEL
LIN {X 0,Y 291.378,Z 421.691,A -85,B 0,C 180,E1 -16717.299,E2 -16717.299} C_VEL
LIN {X 0,Y 291.455,Z 421.682,A -85,B 0,C 180,E1 -16720.269,E2 -16720.269} C_VEL
LIN {X 0,Y 291.552,Z 421.67,A -85,B 0,C 180,E1 -16724.623,E2 -16724.623} C_VEL
LIN {X 0,Y 291.532,Z 421.671,A -85,B 0,C 180,E1 -16728.88,E2 -16728.88} C_VEL
LIN {X 0,Y 291.706,Z 421.647,A -85,B 0,C 180,E1 -16731.688,E2 -16731.688} C_VEL
LIN {X 0,Y 291.626,Z 421.661,A -85,B 0,C 180,E1 -16734.467,E2 -16734.467} C_VEL
LIN {X 0,Y 291.885,Z 421.624,A -85,B 0,C 180,E1 -16738.62,E2 -16738.62} C_VEL
LIN {X 0,Y 291.884,Z 421.614,A -85,B 0,C 180,E1 -16741.379,E2 -16741.379} C_VEL
LIN {X 0,Y 291.741,Z 421.643,A -85,B 0,C 180,E1 -16746.917,E2 -16746.917} C_VEL
LIN {X 0,Y 291.624,Z 421.656,A -85,B 0,C 180,E1 -16749.711,E2 -16749.711} C_VEL
LIN {X 0,Y 291.516,Z 421.673,A -85,B 0,C 180,E1 -16753.95,E2 -16753.95} C_VEL
LIN {X 0,Y 291.481,Z 421.675,A -85,B 0,C 180,E1 -16756.817,E2 -16756.817} C_VEL
LIN {X 0,Y 291.445,Z 421.68,A -85,B 0,C 180,E1 -16759.874,E2 -16759.874} C_VEL
LIN {X 0,Y 291.394,Z 421.685,A -85,B 0,C 180,E1 -16764.205,E2 -16764.205} C_VEL
LIN {X 0,Y 291.416,Z 421.683,A -85,B 0,C 180,E1 -16767.271,E2 -16767.271} C_VEL
LIN {X 0,Y 291.333,Z 421.694,A -85,B 0,C 180,E1 -16770.436,E2 -16770.436} C_VEL
LIN {X 0,Y 291.339,Z 421.696,A -85,B 0,C 180,E1 -16773.698,E2 -16773.698} C_VEL
LIN {X 0,Y 291.399,Z 421.686,A -85,B 0,C 180,E1 -16777.261,E2 -16777.261} C_VEL
LIN {X 0,Y 291.4,Z 421.684,A -85,B 0,C 180,E1 -16780.63,E2 -16780.63} C_VEL
LIN {X 0,Y 291.401,Z 421.685,A -85,B 0,C 180,E1 -16784.379,E2 -16784.379} C_VEL
LIN {X 0,Y 291.385,Z 421.687,A -85,B 0,C 180,E1 -16788.39,E2 -16788.39} C_VEL
LIN {X 0,Y 291.382,Z 421.689,A -85,B 0,C 180,E1 -16791.164,E2 -16791.164} C_VEL
LIN {X 0,Y 291.38,Z 421.688,A -85,B 0,C 180,E1 -16794.63,E2 -16794.63} C_VEL
LIN {X 0,Y 291.366,Z 421.691,A -85,B 0,C 180,E1 -16797.951,E2 -16797.951} C_VEL
LIN {X 0,Y 291.38,Z 421.691,A -85,B 0,C 180,E1 -16801.159,E2 -16801.159} C_VEL
LIN {X 0,Y 291.44,Z 421.682,A -85,B 0,C 180,E1 -16804.542,E2 -16804.542} C_VEL
LIN {X 0,Y 292.362,Z 424.37,A -85,B 0,C 180,E1 -16804.706,E2 -16804.706} C_VEL
LIN {X 0,Y 297.384,Z 434.635,A -85,B 0,C 180,E1 -16805.488,E2 -16805.488} C_VEL
LIN {X 0,Y 302.24,Z 442.721,A -85,B 0,C 180,E1 -16806.287,E2 -16806.287} C_VEL
LIN {X 0,Y 308.22,Z 450.882,A -85,B 0,C 180,E1 -16807.268,E2 -16807.268} C_VEL
LIN {X 0,Y 315.319,Z 459.724,A -85,B 0,C 180,E1 -16808.539,E2 -16808.539} C_VEL
LIN {X 0,Y 321.878,Z 467.302,A -85,B 0,C 180,E1 -16809.861,E2 -16809.861} C_VEL
LIN {X 0,Y 328.278,Z 474.214,A -85,B 0,C 180,E1 -16811.269,E2 -16811.269} C_VEL
LIN {X 0,Y 334.944,Z 481.092,A -85,B 0,C 180,E1 -16812.918,E2 -16812.918} C_VEL
LIN {X 0,Y 340.635,Z 486.518,A -85,B 0,C 180,E1 -16814.442,E2 -16814.442} C_VEL
LIN {X 0,Y 345.257,Z 490.952,A -85,B 0,C 180,E1 -16815.862,E2 -16815.862} C_VEL
LIN {X 0,Y 350.245,Z 495.577,A -85,B 0,C 180,E1 -16817.574,E2 -16817.574} C_VEL
LIN {X 0,Y 354.374,Z 498.99,A -85,B 0,C 180,E1 -16819.134,E2 -16819.134} C_VEL
LIN {X 0,Y 356.732,Z 500.579,A -85,B 0,C 180,E1 -16820.076,E2 -16820.076} C_VEL
LIN {X 0,Y 360.385,Z 504.318,A -85,B 0,C 180,E1 -16822.154,E2 -16822.154} C_VEL
LIN {X 0,Y 362.202,Z 505.818,A -85,B 0,C 180,E1 -16823.315,E2 -16823.315} C_VEL
LIN {X 0,Y 363.799,Z 506.935,A -85,B 0,C 180,E1 -16824.457,E2 -16824.457} C_VEL
LIN {X 0,Y 366.168,Z 508.045,A -85,B 0,C 180,E1 -16826.413,E2 -16826.413} C_VEL
LIN {X 0,Y 367.432,Z 508.382,A -85,B 0,C 180,E1 -16827.808,E2 -16827.808} C_VEL
LIN {X 0,Y 368.04,Z 508.493,A -85,B 0,C 180,E1 -16828.906,E2 -16828.906} C_VEL
LIN {X 0,Y 368.211,Z 508.555,A -85,B 0,C 180,E1 -16830,E2 -16830} C_VEL
LIN {X 0,Y 368.046,Z 508.47,A -85,B 0,C 180,E1 -16831.094,E2 -16831.094} C_VEL
LIN {X 0,Y 367.404,Z 508.39,A -85,B 0,C 180,E1 -16832.193,E2 -16832.193} C_VEL
LIN {X 0,Y 366.176,Z 508.013,A -85,B 0,C 180,E1 -16833.607,E2 -16833.607} C_VEL
LIN {X 0,Y 363.795,Z 506.973,A -85,B 0,C 180,E1 -16835.543,E2 -16835.543} C_VEL
LIN {X 0,Y 361.317,Z 505.153,A -85,B 0,C 180,E1 -16837.257,E2 -16837.257} C_VEL
LIN {X 0,Y 358.418,Z 502.314,A -85,B 0,C 180,E1 -16839.025,E2 -16839.025} C_VEL
LIN {X 0,Y 356.018,Z 500.058,A -85,B 0,C 180,E1 -16840.234,E2 -16840.234} C_VEL
LIN {X 0,Y 351.843,Z 496.988,A -85,B 0,C 180,E1 -16841.832,E2 -16841.832} C_VEL
LIN {X 0,Y 347.035,Z 492.421,A -85,B 0,C 180,E1 -16843.576,E2 -16843.576} C_VEL
LIN {X 0,Y 342.126,Z 488.07,A -85,B 0,C 180,E1 -16845.102,E2 -16845.102} C_VEL
LIN {X 0,Y 337.197,Z 483.218,A -85,B 0,C 180,E1 -16846.517,E2 -16846.517} C_VEL
LIN {X 0,Y 329.633,Z 475.624,A -85,B 0,C 180,E1 -16848.424,E2 -16848.424} C_VEL
LIN {X 0,Y 321.893,Z 467.314,A -85,B 0,C 180,E1 -16850.146,E2 -16850.146} C_VEL
LIN {X 0,Y 315.308,Z 459.696,A -85,B 0,C 180,E1 -16851.458,E2 -16851.458} C_VEL
LIN {X 0,Y 308.224,Z 450.85,A -85,B 0,C 180,E1 -16852.734,E2 -16852.734} C_VEL
LIN {X 0,Y 301.383,Z 441.279,A -85,B 0,C 180,E1 -16853.86,E2 -16853.86} C_VEL
LIN {X 0,Y 296.705,Z 433.487,A -85,B 0,C 180,E1 -16854.62,E2 -16854.62} C_VEL
LIN {X 0,Y 291.63,Z 422.718,A -85,B 0,C 180,E1 -16855.407,E2 -16855.407} C_VEL
LIN {X 0,Y 291.445,Z 421.681,A -85,B 0,C 180,E1 -16855.487,E2 -16855.487} C_VEL
LIN {X 0,Y 291.383,Z 421.688,A -85,B 0,C 180,E1 -16859.74,E2 -16859.74} C_VEL
LIN {X 0,Y 291.341,Z 421.693,A -85,B 0,C 180,E1 -16863.699,E2 -16863.699} C_VEL
LIN {X 0,Y 291.401,Z 421.685,A -85,B 0,C 180,E1 -16867.262,E2 -16867.262} C_VEL
LIN {X 0,Y 291.401,Z 421.688,A -85,B 0,C 180,E1 -16870.631,E2 -16870.631} C_VEL
LIN {X 0,Y 291.349,Z 421.695,A -85,B 0,C 180,E1 -16874.39,E2 -16874.39} C_VEL
LIN {X 0,Y 291.327,Z 421.697,A -85,B 0,C 180,E1 -16878.404,E2 -16878.404} C_VEL
LIN {X 0,Y 291.361,Z 421.689,A -85,B 0,C 180,E1 -16881.161,E2 -16881.161} C_VEL
LIN {X 0,Y 291.382,Z 421.689,A -85,B 0,C 180,E1 -16884.63,E2 -16884.63} C_VEL
LIN {X 0,Y 291.372,Z 421.692,A -85,B 0,C 180,E1 -16887.952,E2 -16887.952} C_VEL
LIN {X 0,Y 291.379,Z 421.687,A -85,B 0,C 180,E1 -16891.159,E2 -16891.159} C_VEL
LIN {X 0,Y 291.413,Z 421.682,A -85,B 0,C 180,E1 -16894.273,E2 -16894.273} C_VEL
LIN {X 0,Y 291.378,Z 421.688,A -85,B 0,C 180,E1 -16897.3,E2 -16897.3} C_VEL
LIN {X 0,Y 291.455,Z 421.679,A -85,B 0,C 180,E1 -16900.271,E2 -16900.271} C_VEL
LIN {X 0,Y 291.552,Z 421.663,A -85,B 0,C 180,E1 -16904.624,E2 -16904.624} C_VEL
LIN {X 0,Y 291.534,Z 421.667,A -85,B 0,C 180,E1 -16908.881,E2 -16908.881} C_VEL
LIN {X 0,Y 291.707,Z 421.649,A -85,B 0,C 180,E1 -16911.689,E2 -16911.689} C_VEL
LIN {X 0,Y 291.628,Z 421.655,A -85,B 0,C 180,E1 -16914.469,E2 -16914.469} C_VEL
LIN {X 0,Y 291.887,Z 421.613,A -85,B 0,C 180,E1 -16918.621,E2 -16918.621} C_VEL
LIN {X 0,Y 291.888,Z 421.624,A -85,B 0,C 180,E1 -16921.38,E2 -16921.38} C_VEL
LIN {X 0,Y 291.745,Z 421.642,A -85,B 0,C 180,E1 -16926.919,E2 -16926.919} C_VEL
LIN {X 0,Y 291.628,Z 421.66,A -85,B 0,C 180,E1 -16929.713,E2 -16929.713} C_VEL
LIN {X 0,Y 291.516,Z 421.671,A -85,B 0,C 180,E1 -16933.876,E2 -16933.876} C_VEL
LIN {X 0,Y 290.882,Z 421.755,A -85,B 0,C 180,E1 -16935.028,E2 -16935.028} C_VEL
LIN {X 0,Y 287.974,Z 422.114,A -85,B 0,C 180,E1 -16936.903,E2 -16936.903} C_VEL
LIN {X 0,Y 285.494,Z 422.421,A -85,B 0,C 180,E1 -16938.425,E2 -16938.425} C_VEL
LIN {X 0,Y 284.453,Z 422.553,A -85,B 0,C 180,E1 -16939.607,E2 -16939.607} C_VEL
LIN {X 0,Y 284.383,Z 422.559,A -85,B 0,C 180,E1 -16940.007,E2 -16940.007} C_VEL
LIN {X 0,Y 284.368,Z 422.563,A -85,B 0,C 180,E1 -16943.876,E2 -16943.876} C_VEL
LIN {X 0,Y 284.394,Z 422.562,A -85,B 0,C 180,E1 -16947.173,E2 -16947.173} C_VEL
LIN {X 0,Y 284.294,Z 422.577,A -85,B 0,C 180,E1 -16951.275,E2 -16951.275} C_VEL
LIN {X 0,Y 284.359,Z 423.001,A -85,B 0,C 180,E1 -16952.939,E2 -16952.939} C_VEL
LIN {X 0,Y 284.668,Z 424.95,A -85,B 0,C 180,E1 -16956.337,E2 -16956.337} C_VEL
LIN {X 0,Y 284.994,Z 427.385,A -85,B 0,C 180,E1 -16960.141,E2 -16960.141} C_VEL
LIN {X 0,Y 285.342,Z 429.81,A -85,B 0,C 180,E1 -16963.603,E2 -16963.603} C_VEL
LIN {X 0,Y 285.538,Z 431.966,A -85,B 0,C 180,E1 -16966.436,E2 -16966.436} C_VEL
LIN {X 0,Y 285.381,Z 434.698,A -85,B 0,C 180,E1 -16969.768,E2 -16969.768} C_VEL
LIN {X 0,Y 284.782,Z 438.153,A -85,B 0,C 180,E1 -16973.681,E2 -16973.681} C_VEL
LIN {X 0,Y 284.176,Z 441.477,A -85,B 0,C 180,E1 -16977.232,E2 -16977.232} C_VEL
LIN {X 0,Y 283.727,Z 444.453,A -85,B 0,C 180,E1 -16980.304,E2 -16980.304} C_VEL
LIN {X 0,Y 283.289,Z 448.243,A -85,B 0,C 180,E1 -16984.112,E2 -16984.112} C_VEL
LIN {X 0,Y 284.661,Z 453.702,A -85,B 0,C 180,E1 -16984.463,E2 -16984.463} C_VEL
LIN {X 0,Y 287.642,Z 465.813,A -85,B 0,C 180,E1 -16985.458,E2 -16985.458} C_VEL
LIN {X 0,Y 289.488,Z 475.696,A -85,B 0,C 180,E1 -16986.4,E2 -16986.4} C_VEL
LIN {X 0,Y 290.673,Z 485.712,A -85,B 0,C 180,E1 -16987.494,E2 -16987.494} C_VEL
LIN {X 0,Y 291.345,Z 494.6,A -85,B 0,C 180,E1 -16988.618,E2 -16988.618} C_VEL
LIN {X 0,Y 290.981,Z 499.901,A -85,B 0,C 180,E1 -16989.315,E2 -16989.315} C_VEL
LIN {X 0,Y 289.189,Z 510.049,A -85,B 0,C 180,E1 -16990.848,E2 -16990.848} C_VEL
LIN {X 0,Y 287.833,Z 518.385,A -85,B 0,C 180,E1 -16992.414,E2 -16992.414} C_VEL
LIN {X 0,Y 286.502,Z 525.397,A -85,B 0,C 180,E1 -16993.98,E2 -16993.98} C_VEL
LIN {X 0,Y 285.273,Z 531.937,A -85,B 0,C 180,E1 -16995.738,E2 -16995.738} C_VEL
LIN {X 0,Y 284.417,Z 536.44,A -85,B 0,C 180,E1 -16997.15,E2 -16997.15} C_VEL
LIN {X 0,Y 283.521,Z 541.937,A -85,B 0,C 180,E1 -16999.286,E2 -16999.286} C_VEL
LIN {X 0,Y 282.881,Z 546.266,A -85,B 0,C 180,E1 -17001.427,E2 -17001.427} C_VEL
LIN {X 0,Y 282.598,Z 548.636,A -85,B 0,C 180,E1 -17002.857,E2 -17002.857} C_VEL
LIN {X 0,Y 282.413,Z 550.735,A -85,B 0,C 180,E1 -17004.523,E2 -17004.523} C_VEL
LIN {X 0,Y 282.35,Z 552.892,A -85,B 0,C 180,E1 -17007.146,E2 -17007.146} C_VEL
LIN {X 0,Y 282.328,Z 553.482,A -85,B 0,C 180,E1 -17008.573,E2 -17008.573} C_VEL
LIN {X 0,Y 282.328,Z 553.482,A -85,B 0,C 180,E1 -17011.426,E2 -17011.426} C_VEL
LIN {X 0,Y 282.35,Z 552.892,A -85,B 0,C 180,E1 -17012.853,E2 -17012.853} C_VEL
LIN {X 0,Y 282.444,Z 550.44,A -85,B 0,C 180,E1 -17015.712,E2 -17015.712} C_VEL
LIN {X 0,Y 282.744,Z 547.486,A -85,B 0,C 180,E1 -17017.857,E2 -17017.857} C_VEL
LIN {X 0,Y 283.259,Z 543.493,A -85,B 0,C 180,E1 -17020.001,E2 -17020.001} C_VEL
LIN {X 0,Y 284.098,Z 538.359,A -85,B 0,C 180,E1 -17022.138,E2 -17022.138} C_VEL
LIN {X 0,Y 285.058,Z 533.095,A -85,B 0,C 180,E1 -17023.909,E2 -17023.909} C_VEL
LIN {X 0,Y 286.226,Z 526.776,A -85,B 0,C 180,E1 -17025.669,E2 -17025.669} C_VEL
LIN {X 0,Y 287.619,Z 519.628,A -85,B 0,C 180,E1 -17027.32,E2 -17027.32} C_VEL
LIN {X 0,Y 288.852,Z 511.973,A -85,B 0,C 180,E1 -17028.806,E2 -17028.806} C_VEL
LIN {X 0,Y 290.313,Z 503.442,A -85,B 0,C 180,E1 -17030.179,E2 -17030.179} C_VEL
LIN {X 0,Y 291.505,Z 495.848,A -85,B 0,C 180,E1 -17031.2,E2 -17031.2} C_VEL
LIN {X 0,Y 290.908,Z 487.625,A -85,B 0,C 180,E1 -17032.269,E2 -17032.269} C_VEL
LIN {X 0,Y 289.85,Z 478.349,A -85,B 0,C 180,E1 -17033.321,E2 -17033.321} C_VEL
LIN {X 0,Y 288.152,Z 468.334,A -85,B 0,C 180,E1 -17034.31,E2 -17034.31} C_VEL
LIN {X 0,Y 285.892,Z 458.386,A -85,B 0,C 180,E1 -17035.162,E2 -17035.162} C_VEL
LIN {X 0,Y 283.369,Z 449.243,A -85,B 0,C 180,E1 -17035.839,E2 -17035.839} C_VEL
LIN {X 0,Y 283.26,Z 448.223,A -85,B 0,C 180,E1 -17035.91,E2 -17035.91} C_VEL
LIN {X 0,Y 283.751,Z 444.244,A -85,B 0,C 180,E1 -17039.9,E2 -17039.9} C_VEL
LIN {X 0,Y 284.185,Z 441.284,A -85,B 0,C 180,E1 -17042.96,E2 -17042.96} C_VEL
LIN {X 0,Y 284.76,Z 438.153,A -85,B 0,C 180,E1 -17046.322,E2 -17046.322} C_VEL
LIN {X 0,Y 285.377,Z 434.689,A -85,B 0,C 180,E1 -17050.231,E2 -17050.231} C_VEL
LIN {X 0,Y 285.536,Z 431.946,A -85,B 0,C 180,E1 -17053.563,E2 -17053.563} C_VEL
LIN {X 0,Y 285.344,Z 429.805,A -85,B 0,C 180,E1 -17056.398,E2 -17056.398} C_VEL
LIN {X 0,Y 284.954,Z 427.211,A -85,B 0,C 180,E1 -17060.114,E2 -17060.114} C_VEL
LIN {X 0,Y 284.589,Z 424.405,A -85,B 0,C 180,E1 -17064.58,E2 -17064.58} C_VEL
LIN {X 0,Y 284.352,Z 422.933,A -85,B 0,C 180,E1 -17067.174,E2 -17067.174} C_VEL
LIN {X 0,Y 284.357,Z 422.566,A -85,B 0,C 180,E1 -17070.375,E2 -17070.375} C_VEL
LIN {X 0,Y 284.375,Z 422.563,A -85,B 0,C 180,E1 -17073.586,E2 -17073.586} C_VEL
LIN {X 0,Y 284.363,Z 422.568,A -85,B 0,C 180,E1 -17076.706,E2 -17076.706} C_VEL
LIN {X 0,Y 284.4,Z 422.559,A -85,B 0,C 180,E1 -17081.261,E2 -17081.261} C_VEL
LIN {X 0,Y 284.488,Z 422.55,A -85,B 0,C 180,E1 -17084.458,E2 -17084.458} C_VEL
LIN {X 0,Y 284.484,Z 422.551,A -85,B 0,C 180,E1 -17088.601,E2 -17088.601} C_VEL
LIN {X 0,Y 284.656,Z 422.525,A -85,B 0,C 180,E1 -17091.48,E2 -17091.48} C_VEL
LIN {X 0,Y 284.597,Z 422.536,A -85,B 0,C 180,E1 -17094.33,E2 -17094.33} C_VEL
LIN {X 0,Y 284.851,Z 422.5,A -85,B 0,C 180,E1 -17098.585,E2 -17098.585} C_VEL
LIN {X 0,Y 284.851,Z 422.489,A -85,B 0,C 180,E1 -17101.413,E2 -17101.413} C_VEL
LIN {X 0,Y 284.693,Z 422.52,A -85,B 0,C 180,E1 -17107.089,E2 -17107.089} C_VEL
LIN {X 0,Y 284.561,Z 422.537,A -85,B 0,C 180,E1 -17109.955,E2 -17109.955} C_VEL
LIN {X 0,Y 284.476,Z 422.547,A -85,B 0,C 180,E1 -17114.302,E2 -17114.302} C_VEL
LIN {X 0,Y 284.42,Z 422.554,A -85,B 0,C 180,E1 -17117.248,E2 -17117.248} C_VEL
LIN {X 0,Y 284.373,Z 422.561,A -85,B 0,C 180,E1 -17120.242,E2 -17120.242} C_VEL
LIN {X 0,Y 284.363,Z 422.564,A -85,B 0,C 180,E1 -17123.875,E2 -17123.875} C_VEL
LIN {X 0,Y 284.391,Z 422.558,A -85,B 0,C 180,E1 -17127.173,E2 -17127.173} C_VEL
LIN {X 0,Y 284.292,Z 422.57,A -85,B 0,C 180,E1 -17131.274,E2 -17131.274} C_VEL
LIN {X 0,Y 284.356,Z 422.564,A -85,B 0,C 180,E1 -17135.354,E2 -17135.354} C_VEL
LIN {X 0,Y 284.332,Z 422.567,A -85,B 0,C 180,E1 -17138.165,E2 -17138.165} C_VEL
LIN {X 0,Y 284.339,Z 422.566,A -85,B 0,C 180,E1 -17142.141,E2 -17142.141} C_VEL
LIN {X 0,Y 284.348,Z 422.564,A -85,B 0,C 180,E1 -17146.208,E2 -17146.208} C_VEL
LIN {X 0,Y 284.346,Z 422.566,A -85,B 0,C 180,E1 -17150.013,E2 -17150.013} C_VEL
LIN {X 0,Y 284.35,Z 422.567,A -85,B 0,C 180,E1 -17153.618,E2 -17153.618} C_VEL
LIN {X 0,Y 284.302,Z 422.572,A -85,B 0,C 180,E1 -17157.19,E2 -17157.19} C_VEL
LIN {X 0,Y 284.354,Z 422.564,A -85,B 0,C 180,E1 -17160.376,E2 -17160.376} C_VEL
LIN {X 0,Y 284.399,Z 422.63,A -85,B 0,C 180,E1 -17163.89,E2 -17163.89} C_VEL
LIN {X 0,Y 285.407,Z 425.446,A -85,B 0,C 180,E1 -17164.067,E2 -17164.067} C_VEL
LIN {X 0,Y 291.692,Z 438.474,A -85,B 0,C 180,E1 -17165.134,E2 -17165.134} C_VEL
LIN {X 0,Y 296.823,Z 447.169,A -85,B 0,C 180,E1 -17166.076,E2 -17166.076} C_VEL
LIN {X 0,Y 303.044,Z 455.718,A -85,B 0,C 180,E1 -17167.196,E2 -17167.196} C_VEL
LIN {X 0,Y 311.272,Z 465.878,A -85,B 0,C 180,E1 -17168.733,E2 -17168.733} C_VEL
LIN {X 0,Y 319.316,Z 474.893,A -85,B 0,C 180,E1 -17170.389,E2 -17170.389} C_VEL
LIN {X 0,Y 325.469,Z 481.461,A -85,B 0,C 180,E1 -17171.823,E2 -17171.823} C_VEL
LIN {X 0,Y 331.94,Z 488.011,A -85,B 0,C 180,E1 -17173.464,E2 -17173.464} C_VEL
LIN {X 0,Y 337.475,Z 493.412,A -85,B 0,C 180,E1 -17175.056,E2 -17175.056} C_VEL
LIN {X 0,Y 341.384,Z 496.888,A -85,B 0,C 180,E1 -17176.268,E2 -17176.268} C_VEL
LIN {X 0,Y 347.039,Z 502.197,A -85,B 0,C 180,E1 -17178.316,E2 -17178.316} C_VEL
LIN {X 0,Y 350.451,Z 504.689,A -85,B 0,C 180,E1 -17179.602,E2 -17179.602} C_VEL
LIN {X 0,Y 353.007,Z 506.92,A -85,B 0,C 180,E1 -17180.836,E2 -17180.836} C_VEL
LIN {X 0,Y 355.031,Z 508.987,A -85,B 0,C 180,E1 -17182.035,E2 -17182.035} C_VEL
LIN {X 0,Y 356.891,Z 510.577,A -85,B 0,C 180,E1 -17183.215,E2 -17183.215} C_VEL
LIN {X 0,Y 359.674,Z 512.406,A -85,B 0,C 180,E1 -17185.221,E2 -17185.221} C_VEL
LIN {X 0,Y 361.359,Z 513.095,A -85,B 0,C 180,E1 -17186.655,E2 -17186.655} C_VEL
LIN {X 0,Y 362.373,Z 513.38,A -85,B 0,C 180,E1 -17187.777,E2 -17187.777} C_VEL
LIN {X 0,Y 363.001,Z 513.518,A -85,B 0,C 180,E1 -17188.891,E2 -17188.891} C_VEL
LIN {X 0,Y 363.193,Z 513.57,A -85,B 0,C 180,E1 -17190,E2 -17190} C_VEL
LIN {X 0,Y 363.006,Z 513.498,A -85,B 0,C 180,E1 -17191.11,E2 -17191.11} C_VEL
LIN {X 0,Y 362.328,Z 513.4,A -85,B 0,C 180,E1 -17192.223,E2 -17192.223} C_VEL
LIN {X 0,Y 361.359,Z 513.081,A -85,B 0,C 180,E1 -17193.345,E2 -17193.345} C_VEL
LIN {X 0,Y 359.674,Z 512.434,A -85,B 0,C 180,E1 -17194.78,E2 -17194.78} C_VEL
LIN {X 0,Y 356.865,Z 510.587,A -85,B 0,C 180,E1 -17196.786,E2 -17196.786} C_VEL
LIN {X 0,Y 354.883,Z 508.895,A -85,B 0,C 180,E1 -17198.04,E2 -17198.04} C_VEL
LIN {X 0,Y 352.069,Z 506.003,A -85,B 0,C 180,E1 -17199.637,E2 -17199.637} C_VEL
LIN {X 0,Y 350.212,Z 504.565,A -85,B 0,C 180,E1 -17200.483,E2 -17200.483} C_VEL
LIN {X 0,Y 345.311,Z 500.596,A -85,B 0,C 180,E1 -17202.335,E2 -17202.335} C_VEL
LIN {X 0,Y 340.461,Z 496.091,A -85,B 0,C 180,E1 -17204.026,E2 -17204.026} C_VEL
LIN {X 0,Y 335.561,Z 491.438,A -85,B 0,C 180,E1 -17205.547,E2 -17205.547} C_VEL
LIN {X 0,Y 328.525,Z 484.622,A -85,B 0,C 180,E1 -17207.427,E2 -17207.427} C_VEL
LIN {X 0,Y 321.297,Z 477.129,A -85,B 0,C 180,E1 -17209.154,E2 -17209.154} C_VEL
LIN {X 0,Y 315.13,Z 470.248,A -85,B 0,C 180,E1 -17210.501,E2 -17210.501} C_VEL
LIN {X 0,Y 308.851,Z 462.916,A -85,B 0,C 180,E1 -17211.732,E2 -17211.732} C_VEL
LIN {X 0,Y 301.669,Z 454.011,A -85,B 0,C 180,E1 -17213.042,E2 -17213.042} C_VEL
LIN {X 0,Y 295.517,Z 444.968,A -85,B 0,C 180,E1 -17214.177,E2 -17214.177} C_VEL
LIN {X 0,Y 290.913,Z 437.075,A -85,B 0,C 180,E1 -17214.998,E2 -17214.998} C_VEL
LIN {X 0,Y 284.563,Z 423.445,A -85,B 0,C 180,E1 -17216.071,E2 -17216.071} C_VEL
LIN {X 0,Y 284.385,Z 422.562,A -85,B 0,C 180,E1 -17216.135,E2 -17216.135} C_VEL
LIN {X 0,Y 284.311,Z 422.571,A -85,B 0,C 180,E1 -17220.099,E2 -17220.099} C_VEL
LIN {X 0,Y 284.302,Z 422.571,A -85,B 0,C 180,E1 -17222.946,E2 -17222.946} C_VEL
LIN {X 0,Y 284.351,Z 422.567,A -85,B 0,C 180,E1 -17226.383,E2 -17226.383} C_VEL
LIN {X 0,Y 284.348,Z 422.566,A -85,B 0,C 180,E1 -17229.987,E2 -17229.987} C_VEL
LIN {X 0,Y 284.314,Z 422.569,A -85,B 0,C 180,E1 -17233.799,E2 -17233.799} C_VEL
LIN {X 0,Y 284.278,Z 422.575,A -85,B 0,C 180,E1 -17238.127,E2 -17238.127} C_VEL
LIN {X 0,Y 284.331,Z 422.569,A -85,B 0,C 180,E1 -17242.275,E2 -17242.275} C_VEL
LIN {X 0,Y 284.32,Z 422.567,A -85,B 0,C 180,E1 -17245.353,E2 -17245.353} C_VEL
LIN {X 0,Y 284.295,Z 422.57,A -85,B 0,C 180,E1 -17248.727,E2 -17248.727} C_VEL
LIN {X 0,Y 284.394,Z 422.558,A -85,B 0,C 180,E1 -17252.827,E2 -17252.827} C_VEL
LIN {X 0,Y 284.363,Z 422.562,A -85,B 0,C 180,E1 -17256.708,E2 -17256.708} C_VEL
LIN {X 0,Y 284.4,Z 422.556,A -85,B 0,C 180,E1 -17261.262,E2 -17261.262} C_VEL
LIN {X 0,Y 284.489,Z 422.543,A -85,B 0,C 180,E1 -17264.46,E2 -17264.46} C_VEL
LIN {X 0,Y 284.485,Z 422.545,A -85,B 0,C 180,E1 -17268.602,E2 -17268.602} C_VEL
LIN {X 0,Y 284.657,Z 422.525,A -85,B 0,C 180,E1 -17271.482,E2 -17271.482} C_VEL
LIN {X 0,Y 284.599,Z 422.531,A -85,B 0,C 180,E1 -17274.332,E2 -17274.332} C_VEL
LIN {X 0,Y 284.853,Z 422.489,A -85,B 0,C 180,E1 -17278.587,E2 -17278.587} C_VEL
LIN {X 0,Y 284.854,Z 422.5,A -85,B 0,C 180,E1 -17281.415,E2 -17281.415} C_VEL
LIN {X 0,Y 284.697,Z 422.521,A -85,B 0,C 180,E1 -17287.091,E2 -17287.091} C_VEL
LIN {X 0,Y 284.565,Z 422.538,A -85,B 0,C 180,E1 -17289.956,E2 -17289.956} C_VEL
LIN {X 0,Y 284.481,Z 422.547,A -85,B 0,C 180,E1 -17294.304,E2 -17294.304} C_VEL
LIN {X 0,Y 284.424,Z 422.558,A -85,B 0,C 180,E1 -17297.249,E2 -17297.249} C_VEL
LIN {X 0,Y 284.383,Z 422.559,A -85,B 0,C 180,E1 -17300.007,E2 -17300.007} C_VEL
LIN {X 0,Y 283.744,Z 422.644,A -85,B 0,C 180,E1 -17301.19,E2 -17301.19} C_VEL
LIN {X 0,Y 280.866,Z 423.003,A -85,B 0,C 180,E1 -17303.115,E2 -17303.115} C_VEL
LIN {X 0,Y 278.414,Z 423.305,A -85,B 0,C 180,E1 -17304.68,E2 -17304.68} C_VEL
LIN {X 0,Y 277.379,Z 423.433,A -85,B 0,C 180,E1 -17305.893,E2 -17305.893} C_VEL
LIN {X 0,Y 277.305,Z 423.441,A -85,B 0,C 180,E1 -17306.304,E2 -17306.304} C_VEL
LIN {X 0,Y 277.273,Z 423.45,A -85,B 0,C 180,E1 -17310.482,E2 -17310.482} C_VEL
LIN {X 0,Y 277.268,Z 423.71,A -85,B 0,C 180,E1 -17312.161,E2 -17312.161} C_VEL
LIN {X 0,Y 277.631,Z 425.785,A -85,B 0,C 180,E1 -17315.899,E2 -17315.899} C_VEL
LIN {X 0,Y 277.874,Z 427.825,A -85,B 0,C 180,E1 -17319.221,E2 -17319.221} C_VEL
LIN {X 0,Y 278.272,Z 430.373,A -85,B 0,C 180,E1 -17322.994,E2 -17322.994} C_VEL
LIN {X 0,Y 278.421,Z 431.826,A -85,B 0,C 180,E1 -17325.027,E2 -17325.027} C_VEL
LIN {X 0,Y 278.503,Z 433.379,A -85,B 0,C 180,E1 -17327.052,E2 -17327.052} C_VEL
LIN {X 0,Y 278.361,Z 435.119,A -85,B 0,C 180,E1 -17329.24,E2 -17329.24} C_VEL
LIN {X 0,Y 277.86,Z 438.001,A -85,B 0,C 180,E1 -17332.625,E2 -17332.625} C_VEL
LIN {X 0,Y 277.277,Z 441.118,A -85,B 0,C 180,E1 -17336.109,E2 -17336.109} C_VEL
LIN {X 0,Y 276.733,Z 444.49,A -85,B 0,C 180,E1 -17339.71,E2 -17339.71} C_VEL
LIN {X 0,Y 276.267,Z 448.136,A -85,B 0,C 180,E1 -17343.412,E2 -17343.412} C_VEL
LIN {X 0,Y 278.453,Z 456.271,A -85,B 0,C 180,E1 -17344.01,E2 -17344.01} C_VEL
LIN {X 0,Y 280.712,Z 465.586,A -85,B 0,C 180,E1 -17344.81,E2 -17344.81} C_VEL
LIN {X 0,Y 282.738,Z 476.306,A -85,B 0,C 180,E1 -17345.881,E2 -17345.881} C_VEL
LIN {X 0,Y 283.83,Z 485.491,A -85,B 0,C 180,E1 -17346.921,E2 -17346.921} C_VEL
LIN {X 0,Y 284.503,Z 494.49,A -85,B 0,C 180,E1 -17348.093,E2 -17348.093} C_VEL
LIN {X 0,Y 284.503,Z 498.336,A -85,B 0,C 180,E1 -17348.632,E2 -17348.632} C_VEL
LIN {X 0,Y 282.484,Z 509.837,A -85,B 0,C 180,E1 -17350.374,E2 -17350.374} C_VEL
LIN {X 0,Y 280.931,Z 518.805,A -85,B 0,C 180,E1 -17352.113,E2 -17352.113} C_VEL
LIN {X 0,Y 279.652,Z 525.185,A -85,B 0,C 180,E1 -17353.577,E2 -17353.577} C_VEL
LIN {X 0,Y 278.371,Z 531.725,A -85,B 0,C 180,E1 -17355.376,E2 -17355.376} C_VEL
LIN {X 0,Y 277.461,Z 536.227,A -85,B 0,C 180,E1 -17356.822,E2 -17356.822} C_VEL
LIN {X 0,Y 276.518,Z 541.725,A -85,B 0,C 180,E1 -17359.011,E2 -17359.011} C_VEL
LIN {X 0,Y 275.836,Z 546.054,A -85,B 0,C 180,E1 -17361.206,E2 -17361.206} C_VEL
LIN {X 0,Y 275.526,Z 548.424,A -85,B 0,C 180,E1 -17362.672,E2 -17362.672} C_VEL
LIN {X 0,Y 275.324,Z 550.758,A -85,B 0,C 180,E1 -17364.585,E2 -17364.585} C_VEL
LIN {X 0,Y 275.261,Z 552.681,A -85,B 0,C 180,E1 -17367.073,E2 -17367.073} C_VEL
LIN {X 0,Y 275.254,Z 553.272,A -85,B 0,C 180,E1 -17368.537,E2 -17368.537} C_VEL
LIN {X 0,Y 275.254,Z 553.272,A -85,B 0,C 180,E1 -17371.463,E2 -17371.463} C_VEL
LIN {X 0,Y 275.261,Z 552.681,A -85,B 0,C 180,E1 -17372.927,E2 -17372.927} C_VEL
LIN {X 0,Y 275.381,Z 550.229,A -85,B 0,C 180,E1 -17375.859,E2 -17375.859} C_VEL
LIN {X 0,Y 275.684,Z 547.274,A -85,B 0,C 180,E1 -17378.06,E2 -17378.06} C_VEL
LIN {X 0,Y 276.245,Z 543.281,A -85,B 0,C 180,E1 -17380.258,E2 -17380.258} C_VEL
LIN {X 0,Y 277.109,Z 538.146,A -85,B 0,C 180,E1 -17382.449,E2 -17382.449} C_VEL
LIN {X 0,Y 278.15,Z 532.883,A -85,B 0,C 180,E1 -17384.261,E2 -17384.261} C_VEL
LIN {X 0,Y 279.352,Z 526.563,A -85,B 0,C 180,E1 -17386.065,E2 -17386.065} C_VEL
LIN {X 0,Y 280.608,Z 520.613,A -85,B 0,C 180,E1 -17387.49,E2 -17387.49} C_VEL
LIN {X 0,Y 281.751,Z 513.68,A -85,B 0,C 180,E1 -17388.921,E2 -17388.921} C_VEL
LIN {X 0,Y 283.245,Z 505.5,A -85,B 0,C 180,E1 -17390.326,E2 -17390.326} C_VEL
LIN {X 0,Y 284.682,Z 496.988,A -85,B 0,C 180,E1 -17391.544,E2 -17391.544} C_VEL
LIN {X 0,Y 284.123,Z 488.21,A -85,B 0,C 180,E1 -17392.736,E2 -17392.736} C_VEL
LIN {X 0,Y 283.045,Z 478.537,A -85,B 0,C 180,E1 -17393.877,E2 -17393.877} C_VEL
LIN {X 0,Y 281.356,Z 468.736,A -85,B 0,C 180,E1 -17394.889,E2 -17394.889} C_VEL
LIN {X 0,Y 279.111,Z 458.745,A -85,B 0,C 180,E1 -17395.784,E2 -17395.784} C_VEL
LIN {X 0,Y 276.352,Z 448.954,A -85,B 0,C 180,E1 -17396.548,E2 -17396.548} C_VEL
LIN {X 0,Y 276.253,Z 448.015,A -85,B 0,C 180,E1 -17396.627,E2 -17396.627} C_VEL
LIN {X 0,Y 276.754,Z 444.248,A -85,B 0,C 180,E1 -17400.522,E2 -17400.522} C_VEL
LIN {X 0,Y 277.26,Z 441.116,A -85,B 0,C 180,E1 -17403.893,E2 -17403.893} C_VEL
LIN {X 0,Y 277.851,Z 437.967,A -85,B 0,C 180,E1 -17407.376,E2 -17407.376} C_VEL
LIN {X 0,Y 278.371,Z 434.892,A -85,B 0,C 180,E1 -17411.026,E2 -17411.026} C_VEL
LIN {X 0,Y 278.499,Z 433.321,A -85,B 0,C 180,E1 -17412.959,E2 -17412.959} C_VEL
LIN {X 0,Y 278.419,Z 431.771,A -85,B 0,C 180,E1 -17415.025,E2 -17415.025} C_VEL
LIN {X 0,Y 278.067,Z 429.028,A -85,B 0,C 180,E1 -17418.917,E2 -17418.917} C_VEL
LIN {X 0,Y 277.684,Z 426.687,A -85,B 0,C 180,E1 -17422.596,E2 -17422.596} C_VEL
LIN {X 0,Y 277.407,Z 424.631,A -85,B 0,C 180,E1 -17426.126,E2 -17426.126} C_VEL
LIN {X 0,Y 277.268,Z 423.709,A -85,B 0,C 180,E1 -17427.839,E2 -17427.839} C_VEL
LIN {X 0,Y 277.288,Z 423.447,A -85,B 0,C 180,E1 -17431.212,E2 -17431.212} C_VEL
LIN {X 0,Y 277.311,Z 423.446,A -85,B 0,C 180,E1 -17434.478,E2 -17434.478} C_VEL
LIN {X 0,Y 277.282,Z 423.447,A -85,B 0,C 180,E1 -17437.654,E2 -17437.654} C_VEL
LIN {X 0,Y 277.342,Z 423.441,A -85,B 0,C 180,E1 -17440.765,E2 -17440.765} C_VEL
LIN {X 0,Y 277.431,Z 423.425,A -85,B 0,C 180,E1 -17445.325,E2 -17445.325} C_VEL
LIN {X 0,Y 277.503,Z 423.416,A -85,B 0,C 180,E1 -17449.788,E2 -17449.788} C_VEL
LIN {X 0,Y 277.649,Z 423.401,A -85,B 0,C 180,E1 -17452.728,E2 -17452.728} C_VEL
LIN {X 0,Y 277.817,Z 423.377,A -85,B 0,C 180,E1 -17458.55,E2 -17458.55} C_VEL
LIN {X 0,Y 277.816,Z 423.364,A -85,B 0,C 180,E1 -17461.449,E2 -17461.449} C_VEL
LIN {X 0,Y 277.648,Z 423.398,A -85,B 0,C 180,E1 -17467.27,E2 -17467.27} C_VEL
LIN {X 0,Y 277.501,Z 423.416,A -85,B 0,C 180,E1 -17470.211,E2 -17470.211} C_VEL
LIN {X 0,Y 277.429,Z 423.423,A -85,B 0,C 180,E1 -17474.674,E2 -17474.674} C_VEL
LIN {X 0,Y 277.339,Z 423.435,A -85,B 0,C 180,E1 -17479.233,E2 -17479.233} C_VEL
LIN {X 0,Y 277.313,Z 423.439,A -85,B 0,C 180,E1 -17484.17,E2 -17484.17} C_VEL
LIN {X 0,Y 277.32,Z 423.44,A -85,B 0,C 180,E1 -17487.505,E2 -17487.505} C_VEL
LIN {X 0,Y 277.266,Z 423.446,A -85,B 0,C 180,E1 -17490.481,E2 -17490.481} C_VEL
LIN {X 0,Y 277.249,Z 423.451,A -85,B 0,C 180,E1 -17493.894,E2 -17493.894} C_VEL
LIN {X 0,Y 277.285,Z 423.445,A -85,B 0,C 180,E1 -17497.465,E2 -17497.465} C_VEL
LIN {X 0,Y 277.261,Z 423.447,A -85,B 0,C 180,E1 -17501.226,E2 -17501.226} C_VEL
LIN {X 0,Y 277.283,Z 423.445,A -85,B 0,C 180,E1 -17505.208,E2 -17505.208} C_VEL
LIN {X 0,Y 277.291,Z 423.445,A -85,B 0,C 180,E1 -17509.494,E2 -17509.494} C_VEL
LIN {X 0,Y 277.285,Z 423.444,A -85,B 0,C 180,E1 -17512.535,E2 -17512.535} C_VEL
LIN {X 0,Y 277.249,Z 423.449,A -85,B 0,C 180,E1 -17516.106,E2 -17516.106} C_VEL
LIN {X 0,Y 277.256,Z 423.451,A -85,B 0,C 180,E1 -17519.539,E2 -17519.539} C_VEL
LIN {X 0,Y 277.334,Z 423.441,A -85,B 0,C 180,E1 -17523.188,E2 -17523.188} C_VEL
LIN {X 0,Y 278.433,Z 426.446,A -85,B 0,C 180,E1 -17523.389,E2 -17523.389} C_VEL
LIN {X 0,Y 284.799,Z 440.022,A -85,B 0,C 180,E1 -17524.557,E2 -17524.557} C_VEL
LIN {X 0,Y 289.244,Z 448.16,A -85,B 0,C 180,E1 -17525.456,E2 -17525.456} C_VEL
LIN {X 0,Y 295.829,Z 457.955,A -85,B 0,C 180,E1 -17526.776,E2 -17526.776} C_VEL
LIN {X 0,Y 304.025,Z 468.235,A -85,B 0,C 180,E1 -17528.41,E2 -17528.41} C_VEL
LIN {X 0,Y 313.413,Z 478.977,A -85,B 0,C 180,E1 -17530.356,E2 -17530.356} C_VEL
LIN {X 0,Y 319.555,Z 485.564,A -85,B 0,C 180,E1 -17531.782,E2 -17531.782} C_VEL
LIN {X 0,Y 325.591,Z 491.701,A -85,B 0,C 180,E1 -17533.293,E2 -17533.293} C_VEL
LIN {X 0,Y 331.454,Z 497.367,A -85,B 0,C 180,E1 -17534.946,E2 -17534.946} C_VEL
LIN {X 0,Y 335.983,Z 501.454,A -85,B 0,C 180,E1 -17536.354,E2 -17536.354} C_VEL
LIN {X 0,Y 340.849,Z 506.086,A -85,B 0,C 180,E1 -17538.101,E2 -17538.101} C_VEL
LIN {X 0,Y 344.329,Z 508.785,A -85,B 0,C 180,E1 -17539.415,E2 -17539.415} C_VEL
LIN {X 0,Y 347.153,Z 511.041,A -85,B 0,C 180,E1 -17540.68,E2 -17540.68} C_VEL
LIN {X 0,Y 349.26,Z 513.172,A -85,B 0,C 180,E1 -17541.903,E2 -17541.903} C_VEL
LIN {X 0,Y 351.165,Z 514.885,A -85,B 0,C 180,E1 -17543.104,E2 -17543.104} C_VEL
LIN {X 0,Y 353.066,Z 516.282,A -85,B 0,C 180,E1 -17544.423,E2 -17544.423} C_VEL
LIN {X 0,Y 354.464,Z 517.051,A -85,B 0,C 180,E1 -17545.451,E2 -17545.451} C_VEL
